LIN {X 0,Y 183.796,Z 363.678,A -85,B 0,C 180,E1 7701.816,E2 7701.816} C_VEL
LIN {X 0,Y 180.44,Z 378.523,A -85,B 0,C 180,E1 7700.122,E2 7700.122} C_VEL
LIN {X 0,Y 176.218,Z 391.784,A -85,B 0,C 180,E1 7698.008,E2 7698.008} C_VEL
LIN {X 0,Y 171.582,Z 403.279,A -85,B 0,C 180,E1 7695.544,E2 7695.544} C_VEL
LIN {X 0,Y 166.647,Z 413.424,A -85,B 0,C 180,E1 7692.682,E2 7692.682} C_VEL
LIN {X 0,Y 161.304,Z 422.653,A -85,B 0,C 180,E1 7689.21,E2 7689.21} C_VEL
LIN {X 0,Y 156.045,Z 430.534,A -85,B 0,C 180,E1 7685.213,E2 7685.213} C_VEL
LIN {X 0,Y 150.742,Z 437.424,A -85,B 0,C 180,E1 7680.268,E2 7680.268} C_VEL
LIN {X 0,Y 146.163,Z 442.505,A -85,B 0,C 180,E1 7674.659,E2 7674.659} C_VEL
LIN {X 0,Y 142.797,Z 445.543,A -85,B 0,C 180,E1 7668.786,E2 7668.786} C_VEL
LIN {X 0,Y 140.665,Z 446.734,A -85,B 0,C 180,E1 7662.726,E2 7662.726} C_VEL
LIN {X 0,Y 139.739,Z 446.152,A -85,B 0,C 180,E1 7656.571,E2 7656.571} C_VEL
LIN {X 0,Y 140.025,Z 443.543,A -85,B 0,C 180,E1 7649.997,E2 7649.997} C_VEL
LIN {X 0,Y 141.478,Z 439.126,A -85,B 0,C 180,E1 7643.912,E2 7643.912} C_VEL
LIN {X 0,Y 143.867,Z 433.071,A -85,B 0,C 180,E1 7638.37,E2 7638.37} C_VEL
LIN {X 0,Y 146.979,Z 425.519,A -85,B 0,C 180,E1 7633.396,E2 7633.396} C_VEL
LIN {X 0,Y 147.344,Z 424.201,A -85,B 0,C 180,E1 7632.625,E2 7632.625} C_VEL
LIN {X 0,Y 145.87,Z 423.422,A -85,B 0,C 180,E1 7631.533,E2 7631.533} C_VEL
LIN {X 0,Y 141.985,Z 433.557,A -85,B 0,C 180,E1 7624.342,E2 7624.342} C_VEL
LIN {X 0,Y 140.16,Z 439.981,A -85,B 0,C 180,E1 7618.095,E2 7618.095} C_VEL
LIN {X 0,Y 139.61,Z 444.799,A -85,B 0,C 180,E1 7611.456,E2 7611.456} C_VEL
LIN {X 0,Y 140.498,Z 447.794,A -85,B 0,C 180,E1 7604.627,E2 7604.627} C_VEL
LIN {X 0,Y 143.009,Z 449.031,A -85,B 0,C 180,E1 7597.807,E2 7597.807} C_VEL
LIN {X 0,Y 146.933,Z 448.501,A -85,B 0,C 180,E1 7591.6,E2 7591.6} C_VEL
LIN {X 0,Y 152.727,Z 446.052,A -85,B 0,C 180,E1 7585.381,E2 7585.381} C_VEL
LIN {X 0,Y 160,Z 441.734,A -85,B 0,C 180,E1 7579.723,E2 7579.723} C_VEL
LIN {X 0,Y 168.194,Z 435.599,A -85,B 0,C 180,E1 7574.811,E2 7574.811} C_VEL
LIN {X 0,Y 176.992,Z 427.833,A -85,B 0,C 180,E1 7570.586,E2 7570.586} C_VEL
LIN {X 0,Y 185.661,Z 418.872,A -85,B 0,C 180,E1 7567.116,E2 7567.116} C_VEL
LIN {X 0,Y 194.986,Z 407.509,A -85,B 0,C 180,E1 7563.936,E2 7563.936} C_VEL
LIN {X 0,Y 203.524,Z 395.312,A -85,B 0,C 180,E1 7561.408,E2 7561.408} C_VEL
LIN {X 0,Y 210.985,Z 382.54,A -85,B 0,C 180,E1 7559.417,E2 7559.417} C_VEL
LIN {X 0,Y 218.224,Z 367.365,A -85,B 0,C 180,E1 7557.637,E2 7557.637} C_VEL
LIN {X 0,Y 224.14,Z 351.874,A -85,B 0,C 180,E1 7556.279,E2 7556.279} C_VEL
LIN {X 0,Y 228.785,Z 335.328,A -85,B 0,C 180,E1 7555.225,E2 7555.225} C_VEL
LIN {X 0,Y 232.053,Z 318.038,A -85,B 0,C 180,E1 7554.464,E2 7554.464} C_VEL
LIN {X 0,Y 241.488,Z 250.304,A -85,B 0,C 180,E1 7552.506,E2 7552.506} C_VEL
LIN {X 0,Y 240.741,Z 246.563,A -85,B 0,C 180,E1 7550.498,E2 7550.498} C_VEL
LIN {X 0,Y 240.162,Z 243.632,A -85,B 0,C 180,E1 7548.351,E2 7548.351} C_VEL
LIN {X 0,Y 239.883,Z 241.404,A -85,B 0,C 180,E1 7545.243,E2 7545.243} C_VEL
LIN {X 0,Y 240.273,Z 241.241,A -85,B 0,C 180,E1 7542.065,E2 7542.065} C_VEL
LIN {X 0,Y 241.515,Z 243.115,A -85,B 0,C 180,E1 7538.635,E2 7538.635} C_VEL
LIN {X 0,Y 242.511,Z 245.708,A -85,B 0,C 180,E1 7536.743,E2 7536.743} C_VEL
LIN {X 0,Y 230.891,Z 333.654,A -85,B 0,C 180,E1 7534.471,E2 7534.471} C_VEL
LIN {X 0,Y 227.213,Z 350.101,A -85,B 0,C 180,E1 7533.868,E2 7533.868} C_VEL
LIN {X 0,Y 224.792,Z 357.503,A -85,B 0,C 180,E1 7533.772,E2 7533.772} C_VEL
LIN {X 0,Y 217.369,Z 373.68,A -85,B 0,C 180,E1 7534.209,E2 7534.209} C_VEL
LIN {X 0,Y 213.861,Z 380.585,A -85,B 0,C 180,E1 7534.095,E2 7534.095} C_VEL
LIN {X 0,Y 212.895,Z 382.52,A -85,B 0,C 180,E1 7533.967,E2 7533.967} C_VEL
LIN {X 0,Y 204.588,Z 398.255,A -85,B 0,C 180,E1 7532.504,E2 7532.504} C_VEL
LIN {X 0,Y 195.17,Z 413.15,A -85,B 0,C 180,E1 7530.568,E2 7530.568} C_VEL
LIN {X 0,Y 184.964,Z 426.922,A -85,B 0,C 180,E1 7528.073,E2 7528.073} C_VEL
LIN {X 0,Y 174.557,Z 439.14,A -85,B 0,C 180,E1 7524.998,E2 7524.998} C_VEL
LIN {X 0,Y 163.56,Z 450.596,A -85,B 0,C 180,E1 7520.932,E2 7520.932} C_VEL
LIN {X 0,Y 153.123,Z 460.494,A -85,B 0,C 180,E1 7515.915,E2 7515.915} C_VEL
LIN {X 0,Y 144.228,Z 468.323,A -85,B 0,C 180,E1 7510.148,E2 7510.148} C_VEL
LIN {X 0,Y 136.834,Z 474.713,A -85,B 0,C 180,E1 7503.235,E2 7503.235} C_VEL
LIN {X 0,Y 131.616,Z 479.56,A -85,B 0,C 180,E1 7495.18,E2 7495.18} C_VEL
LIN {X 0,Y 129.261,Z 482.628,A -85,B 0,C 180,E1 7486.433,E2 7486.433} C_VEL
LIN {X 0,Y 129.758,Z 483.716,A -85,B 0,C 180,E1 7477.976,E2 7477.976} C_VEL
LIN {X 0,Y 131.875,Z 483.304,A -85,B 0,C 180,E1 7470.438,E2 7470.438} C_VEL
LIN {X 0,Y 130.994,Z 483.773,A -85,B 0,C 180,E1 7466.941,E2 7466.941} C_VEL
LIN {X 0,Y 129.415,Z 483.078,A -85,B 0,C 180,E1 7460.217,E2 7460.217} C_VEL
LIN {X 0,Y 129.295,Z 480.56,A -85,B 0,C 180,E1 7453.378,E2 7453.378} C_VEL
LIN {X 0,Y 130.92,Z 476.166,A -85,B 0,C 180,E1 7446.605,E2 7446.605} C_VEL
LIN {X 0,Y 134.304,Z 469.671,A -85,B 0,C 180,E1 7440.084,E2 7440.084} C_VEL
LIN {X 0,Y 138.579,Z 462.091,A -85,B 0,C 180,E1 7434.75,E2 7434.75} C_VEL
LIN {X 0,Y 143.545,Z 453.197,A -85,B 0,C 180,E1 7430.152,E2 7430.152} C_VEL
LIN {X 0,Y 149.389,Z 441.861,A -85,B 0,C 180,E1 7425.893,E2 7425.893} C_VEL
LIN {X 0,Y 155.141,Z 429.09,A -85,B 0,C 180,E1 7422.45,E2 7422.45} C_VEL
LIN {X 0,Y 159.866,Z 416.561,A -85,B 0,C 180,E1 7419.995,E2 7419.995} C_VEL
LIN {X 0,Y 163.873,Z 403.35,A -85,B 0,C 180,E1 7418.092,E2 7418.092} C_VEL
LIN {X 0,Y 167.255,Z 387.828,A -85,B 0,C 180,E1 7416.541,E2 7416.541} C_VEL
LIN {X 0,Y 169.352,Z 371.857,A -85,B 0,C 180,E1 7415.588,E2 7415.588} C_VEL
LIN {X 0,Y 170.942,Z 353.783,A -85,B 0,C 180,E1 7414.832,E2 7414.832} C_VEL
LIN {X 0,Y 173.502,Z 335.522,A -85,B 0,C 180,E1 7413.757,E2 7413.757} C_VEL
LIN {X 0,Y 181.035,Z 244.738,A -85,B 0,C 180,E1 7410.511,E2 7410.511} C_VEL
LIN {X 0,Y 191.3,Z 201.884,A -85,B 0,C 180,E1 7407.552,E2 7407.552} C_VEL
LIN {X 0,Y 189.274,Z 188.28,A -85,B 0,C 180,E1 7402.682,E2 7402.682} C_VEL
LIN {X 0,Y 187.949,Z 177.866,A -85,B 0,C 180,E1 7398.132,E2 7398.132} C_VEL
LIN {X 0,Y 187.052,Z 175.913,A -85,B 0,C 180,E1 7396.138,E2 7396.138} C_VEL
LIN {X 0,Y 184.12,Z 171.648,A -85,B 0,C 180,E1 7387.174,E2 7387.174} C_VEL
LIN {X 0,Y 183.556,Z 171.776,A -85,B 0,C 180,E1 7383.747,E2 7383.747} C_VEL
LIN {X 0,Y 183.965,Z 175.013,A -85,B 0,C 180,E1 7375.323,E2 7375.323} C_VEL
LIN {X 0,Y 185.238,Z 179.369,A -85,B 0,C 180,E1 7370.367,E2 7370.367} C_VEL
LIN {X 0,Y 186.45,Z 183.613,A -85,B 0,C 180,E1 7366.667,E2 7366.667} C_VEL
LIN {X 0,Y 188.095,Z 189.403,A -85,B 0,C 180,E1 7362.681,E2 7362.681} C_VEL
LIN {X 0,Y 189.901,Z 196.74,A -85,B 0,C 180,E1 7358.697,E2 7358.697} C_VEL
LIN {X 0,Y 191.572,Z 205.206,A -85,B 0,C 180,E1 7354.99,E2 7354.99} C_VEL
LIN {X 0,Y 192.499,Z 212.026,A -85,B 0,C 180,E1 7352.541,E2 7352.541} C_VEL
LIN {X 0,Y 188.599,Z 232.595,A -85,B 0,C 180,E1 7349.437,E2 7349.437} C_VEL
LIN {X 0,Y 188.915,Z 240.844,A -85,B 0,C 180,E1 7348.727,E2 7348.727} C_VEL
LIN {X 0,Y 182.567,Z 320.837,A -85,B 0,C 180,E1 7346.205,E2 7346.205} C_VEL
LIN {X 0,Y 180.809,Z 349.598,A -85,B 0,C 180,E1 7344.905,E2 7344.905} C_VEL
LIN {X 0,Y 178.761,Z 364.13,A -85,B 0,C 180,E1 7343.782,E2 7343.782} C_VEL
LIN {X 0,Y 175.424,Z 378.468,A -85,B 0,C 180,E1 7342.163,E2 7342.163} C_VEL
LIN {X 0,Y 171.236,Z 391.377,A -85,B 0,C 180,E1 7340.155,E2 7340.155} C_VEL
LIN {X 0,Y 166.342,Z 403.249,A -85,B 0,C 180,E1 7337.67,E2 7337.67} C_VEL
LIN {X 0,Y 160.841,Z 414.076,A -85,B 0,C 180,E1 7334.62,E2 7334.62} C_VEL
LIN {X 0,Y 155.136,Z 423.474,A -85,B 0,C 180,E1 7331.054,E2 7331.054} C_VEL
LIN {X 0,Y 149.57,Z 431.381,A -85,B 0,C 180,E1 7326.983,E2 7326.983} C_VEL
LIN {X 0,Y 143.88,Z 438.33,A -85,B 0,C 180,E1 7321.876,E2 7321.876} C_VEL
LIN {X 0,Y 139.217,Z 443.189,A -85,B 0,C 180,E1 7316.438,E2 7316.438} C_VEL
LIN {X 0,Y 135.535,Z 446.37,A -85,B 0,C 180,E1 7310.46,E2 7310.46} C_VEL
LIN {X 0,Y 133.01,Z 447.81,A -85,B 0,C 180,E1 7303.915,E2 7303.915} C_VEL
LIN {X 0,Y 131.832,Z 447.296,A -85,B 0,C 180,E1 7296.967,E2 7296.967} C_VEL
LIN {X 0,Y 132.082,Z 444.737,A -85,B 0,C 180,E1 7289.997,E2 7289.997} C_VEL
LIN {X 0,Y 133.597,Z 440.371,A -85,B 0,C 180,E1 7283.551,E2 7283.551} C_VEL
LIN {X 0,Y 136.123,Z 434.384,A -85,B 0,C 180,E1 7277.698,E2 7277.698} C_VEL
LIN {X 0,Y 139.286,Z 427.144,A -85,B 0,C 180,E1 7272.609,E2 7272.609} C_VEL
LIN {X 0,Y 137.358,Z 426.181,A -85,B 0,C 180,E1 7271.141,E2 7271.141} C_VEL
LIN {X 0,Y 133.913,Z 434.986,A -85,B 0,C 180,E1 7264.335,E2 7264.335} C_VEL
LIN {X 0,Y 132.028,Z 441.741,A -85,B 0,C 180,E1 7257.207,E2 7257.207} C_VEL
LIN {X 0,Y 131.693,Z 446.225,A -85,B 0,C 180,E1 7250.372,E2 7250.372} C_VEL
LIN {X 0,Y 132.906,Z 449.118,A -85,B 0,C 180,E1 7243.132,E2 7243.132} C_VEL
LIN {X 0,Y 135.887,Z 450.266,A -85,B 0,C 180,E1 7235.96,E2 7235.96} C_VEL
LIN {X 0,Y 140.709,Z 449.5,A -85,B 0,C 180,E1 7229.066,E2 7229.066} C_VEL
LIN {X 0,Y 147.342,Z 446.84,A -85,B 0,C 180,E1 7222.642,E2 7222.642} C_VEL
LIN {X 0,Y 154.93,Z 442.571,A -85,B 0,C 180,E1 7217.221,E2 7217.221} C_VEL
LIN {X 0,Y 163.752,Z 436.36,A -85,B 0,C 180,E1 7212.318,E2 7212.318} C_VEL
LIN {X 0,Y 173.27,Z 428.382,A -85,B 0,C 180,E1 7208.078,E2 7208.078} C_VEL
LIN {X 0,Y 182.575,Z 419.158,A -85,B 0,C 180,E1 7204.633,E2 7204.633} C_VEL
LIN {X 0,Y 192.056,Z 408.086,A -85,B 0,C 180,E1 7201.643,E2 7201.643} C_VEL
LIN {X 0,Y 201.142,Z 395.526,A -85,B 0,C 180,E1 7199.146,E2 7199.146} C_VEL
LIN {X 0,Y 209.233,Z 382.045,A -85,B 0,C 180,E1 7197.151,E2 7197.151} C_VEL
LIN {X 0,Y 216.649,Z 366.908,A -85,B 0,C 180,E1 7195.475,E2 7195.475} C_VEL
LIN {X 0,Y 222.539,Z 351.55,A -85,B 0,C 180,E1 7194.211,E2 7194.211} C_VEL
LIN {X 0,Y 227.291,Z 334.726,A -85,B 0,C 180,E1 7193.203,E2 7193.203} C_VEL
LIN {X 0,Y 230.555,Z 317.53,A -85,B 0,C 180,E1 7192.492,E2 7192.492} C_VEL
LIN {X 0,Y 239.48,Z 255.386,A -85,B 0,C 180,E1 7190.75,E2 7190.75} C_VEL
LIN {X 0,Y 238.842,Z 251.44,A -85,B 0,C 180,E1 7188.041,E2 7188.041} C_VEL
LIN {X 0,Y 238.655,Z 249.244,A -85,B 0,C 180,E1 7184.945,E2 7184.945} C_VEL
LIN {X 0,Y 239.067,Z 249.206,A -85,B 0,C 180,E1 7181.972,E2 7181.972} C_VEL
LIN {X 0,Y 240.17,Z 250.984,A -85,B 0,C 180,E1 7178.881,E2 7178.881} C_VEL
LIN {X 0,Y 240.303,Z 251.671,A -85,B 0,C 180,E1 7178.473,E2 7178.473} C_VEL
LIN {X 0,Y 229.224,Z 332.504,A -85,B 0,C 180,E1 7176.449,E2 7176.449} C_VEL
LIN {X 0,Y 224.869,Z 350.985,A -85,B 0,C 180,E1 7175.796,E2 7175.796} C_VEL
LIN {X 0,Y 219.099,Z 368.129,A -85,B 0,C 180,E1 7174.941,E2 7174.941} C_VEL
LIN {X 0,Y 212.895,Z 382.52,A -85,B 0,C 180,E1 7173.967,E2 7173.967} C_VEL
LIN {X 0,Y 209.155,Z 389.39,A -85,B 0,C 180,E1 7173.651,E2 7173.651} C_VEL
LIN {X 0,Y 198.862,Z 403.987,A -85,B 0,C 180,E1 7173.579,E2 7173.579} C_VEL
LIN {X 0,Y 194.314,Z 410.036,A -85,B 0,C 180,E1 7173.203,E2 7173.203} C_VEL
LIN {X 0,Y 193.113,Z 411.695,A -85,B 0,C 180,E1 7172.995,E2 7172.995} C_VEL
LIN {X 0,Y 183.25,Z 424.637,A -85,B 0,C 180,E1 7170.812,E2 7170.812} C_VEL
LIN {X 0,Y 172.328,Z 437.018,A -85,B 0,C 180,E1 7167.901,E2 7167.901} C_VEL
LIN {X 0,Y 160.652,Z 448.602,A -85,B 0,C 180,E1 7164.01,E2 7164.01} C_VEL
LIN {X 0,Y 150.025,Z 458.061,A -85,B 0,C 180,E1 7159.447,E2 7159.447} C_VEL
LIN {X 0,Y 139.614,Z 466.571,A -85,B 0,C 180,E1 7153.437,E2 7153.437} C_VEL
LIN {X 0,Y 131.208,Z 473.061,A -85,B 0,C 180,E1 7146.473,E2 7146.473} C_VEL
LIN {X 0,Y 124.945,Z 478,A -85,B 0,C 180,E1 7138.177,E2 7138.177} C_VEL
LIN {X 0,Y 121.653,Z 481.153,A -85,B 0,C 180,E1 7129.062,E2 7129.062} C_VEL
LIN {X 0,Y 121.494,Z 482.433,A -85,B 0,C 180,E1 7119.955,E2 7119.955} C_VEL
LIN {X 0,Y 123.521,Z 481.958,A -85,B 0,C 180,E1 7111.859,E2 7111.859} C_VEL
LIN {X 0,Y 123.844,Z 482.358,A -85,B 0,C 180,E1 7109.541,E2 7109.541} C_VEL
LIN {X 0,Y 121.921,Z 482.518,A -85,B 0,C 180,E1 7102.938,E2 7102.938} C_VEL
LIN {X 0,Y 121.188,Z 480.901,A -85,B 0,C 180,E1 7095.673,E2 7095.673} C_VEL
LIN {X 0,Y 122.25,Z 477.411,A -85,B 0,C 180,E1 7088.409,E2 7088.409} C_VEL
LIN {X 0,Y 124.954,Z 472.42,A -85,B 0,C 180,E1 7081.833,E2 7081.833} C_VEL
LIN {X 0,Y 129.243,Z 465.518,A -85,B 0,C 180,E1 7075.62,E2 7075.62} C_VEL
LIN {X 0,Y 134.533,Z 457.053,A -85,B 0,C 180,E1 7070.276,E2 7070.276} C_VEL
LIN {X 0,Y 139.88,Z 448.042,A -85,B 0,C 180,E1 7066.109,E2 7066.109} C_VEL
LIN {X 0,Y 145.909,Z 436.717,A -85,B 0,C 180,E1 7062.267,E2 7062.267} C_VEL
LIN {X 0,Y 151.602,Z 424.223,A -85,B 0,C 180,E1 7059.206,E2 7059.206} C_VEL
LIN {X 0,Y 156.414,Z 411.487,A -85,B 0,C 180,E1 7056.932,E2 7056.932} C_VEL
LIN {X 0,Y 160.678,Z 396.975,A -85,B 0,C 180,E1 7055.092,E2 7055.092} C_VEL
LIN {X 0,Y 163.805,Z 381.683,A -85,B 0,C 180,E1 7053.824,E2 7053.824} C_VEL
LIN {X 0,Y 165.534,Z 365.855,A -85,B 0,C 180,E1 7053.019,E2 7053.019} C_VEL
LIN {X 0,Y 174.621,Z 255.346,A -85,B 0,C 180,E1 7049.006,E2 7049.006} C_VEL
LIN {X 0,Y 187.079,Z 205.346,A -85,B 0,C 180,E1 7045.558,E2 7045.558} C_VEL
LIN {X 0,Y 185.622,Z 193.516,A -85,B 0,C 180,E1 7041.155,E2 7041.155} C_VEL
LIN {X 0,Y 184.931,Z 184.749,A -85,B 0,C 180,E1 7037.218,E2 7037.218} C_VEL
LIN {X 0,Y 184.057,Z 183.174,A -85,B 0,C 180,E1 7035.437,E2 7035.437} C_VEL
LIN {X 0,Y 181.483,Z 179.183,A -85,B 0,C 180,E1 7026.961,E2 7026.961} C_VEL
LIN {X 0,Y 180.96,Z 179.369,A -85,B 0,C 180,E1 7023.801,E2 7023.801} C_VEL
LIN {X 0,Y 181.161,Z 182.294,A -85,B 0,C 180,E1 7015.885,E2 7015.885} C_VEL
LIN {X 0,Y 181.959,Z 186.551,A -85,B 0,C 180,E1 7010.83,E2 7010.83} C_VEL
LIN {X 0,Y 183.046,Z 190.826,A -85,B 0,C 180,E1 7007.058,E2 7007.058} C_VEL
LIN {X 0,Y 184.708,Z 197.276,A -85,B 0,C 180,E1 7002.678,E2 7002.678} C_VEL
LIN {X 0,Y 186.345,Z 205.722,A -85,B 0,C 180,E1 6998.27,E2 6998.27} C_VEL
LIN {X 0,Y 187.814,Z 215.098,A -85,B 0,C 180,E1 6994.454,E2 6994.454} C_VEL
LIN {X 0,Y 187.708,Z 216.611,A -85,B 0,C 180,E1 6994.1,E2 6994.1} C_VEL
LIN {X 0,Y 184.249,Z 233.796,A -85,B 0,C 180,E1 6991.496,E2 6991.496} C_VEL
LIN {X 0,Y 184.478,Z 242.195,A -85,B 0,C 180,E1 6990.756,E2 6990.756} C_VEL
LIN {X 0,Y 177.922,Z 321.341,A -85,B 0,C 180,E1 6988.269,E2 6988.269} C_VEL
LIN {X 0,Y 175.985,Z 350.749,A -85,B 0,C 180,E1 6986.926,E2 6986.926} C_VEL
LIN {X 0,Y 173.789,Z 365.423,A -85,B 0,C 180,E1 6985.78,E2 6985.78} C_VEL
LIN {X 0,Y 170.243,Z 379.828,A -85,B 0,C 180,E1 6984.138,E2 6984.138} C_VEL
LIN {X 0,Y 165.892,Z 392.552,A -85,B 0,C 180,E1 6982.139,E2 6982.139} C_VEL
LIN {X 0,Y 160.777,Z 404.347,A -85,B 0,C 180,E1 6979.647,E2 6979.647} C_VEL
LIN {X 0,Y 154.671,Z 415.715,A -85,B 0,C 180,E1 6976.382,E2 6976.382} C_VEL
LIN {X 0,Y 148.189,Z 425.663,A -85,B 0,C 180,E1 6972.427,E2 6972.427} C_VEL
LIN {X 0,Y 142.025,Z 433.686,A -85,B 0,C 180,E1 6967.954,E2 6967.954} C_VEL
LIN {X 0,Y 136.352,Z 440.055,A -85,B 0,C 180,E1 6962.859,E2 6962.859} C_VEL
LIN {X 0,Y 131.47,Z 444.731,A -85,B 0,C 180,E1 6957.145,E2 6957.145} C_VEL
LIN {X 0,Y 127.541,Z 447.754,A -85,B 0,C 180,E1 6950.653,E2 6950.653} C_VEL
LIN {X 0,Y 125.019,Z 448.929,A -85,B 0,C 180,E1 6943.879,E2 6943.879} C_VEL
LIN {X 0,Y 123.898,Z 448.331,A -85,B 0,C 180,E1 6936.949,E2 6936.949} C_VEL
LIN {X 0,Y 124.137,Z 445.923,A -85,B 0,C 180,E1 6929.996,E2 6929.996} C_VEL
LIN {X 0,Y 125.722,Z 441.617,A -85,B 0,C 180,E1 6923.145,E2 6923.145} C_VEL
LIN {X 0,Y 128.172,Z 436.197,A -85,B 0,C 180,E1 6917.38,E2 6917.38} C_VEL
LIN {X 0,Y 131.024,Z 429.999,A -85,B 0,C 180,E1 6912.537,E2 6912.537} C_VEL
LIN {X 0,Y 128.849,Z 428.917,A -85,B 0,C 180,E1 6910.699,E2 6910.699} C_VEL
LIN {X 0,Y 125.198,Z 438.327,A -85,B 0,C 180,E1 6902.403,E2 6902.403} C_VEL
LIN {X 0,Y 123.794,Z 444.268,A -85,B 0,C 180,E1 6895.005,E2 6895.005} C_VEL
LIN {X 0,Y 124.027,Z 448.452,A -85,B 0,C 180,E1 6887.373,E2 6887.373} C_VEL
LIN {X 0,Y 126.048,Z 450.835,A -85,B 0,C 180,E1 6879.692,E2 6879.692} C_VEL
LIN {X 0,Y 130.142,Z 451.423,A -85,B 0,C 180,E1 6872.014,E2 6872.014} C_VEL
LIN {X 0,Y 135.91,Z 450.205,A -85,B 0,C 180,E1 6865.187,E2 6865.187} C_VEL
LIN {X 0,Y 143.046,Z 447.274,A -85,B 0,C 180,E1 6859.18,E2 6859.18} C_VEL
LIN {X 0,Y 152.158,Z 442.224,A -85,B 0,C 180,E1 6853.451,E2 6853.451} C_VEL
LIN {X 0,Y 161.852,Z 435.547,A -85,B 0,C 180,E1 6848.718,E2 6848.718} C_VEL
LIN {X 0,Y 172.127,Z 426.993,A -85,B 0,C 180,E1 6844.665,E2 6844.665} C_VEL
LIN {X 0,Y 182.034,Z 417.242,A -85,B 0,C 180,E1 6841.414,E2 6841.414} C_VEL
LIN {X 0,Y 191.295,Z 406.5,A -85,B 0,C 180,E1 6838.803,E2 6838.803} C_VEL
LIN {X 0,Y 200.339,Z 394.02,A -85,B 0,C 180,E1 6836.551,E2 6836.551} C_VEL
LIN {X 0,Y 208.268,Z 380.879,A -85,B 0,C 180,E1 6834.767,E2 6834.767} C_VEL
LIN {X 0,Y 215.454,Z 366.393,A -85,B 0,C 180,E1 6833.28,E2 6833.28} C_VEL
LIN {X 0,Y 221.477,Z 350.826,A -85,B 0,C 180,E1 6832.086,E2 6832.086} C_VEL
LIN {X 0,Y 226.316,Z 333.886,A -85,B 0,C 180,E1 6831.14,E2 6831.14} C_VEL
LIN {X 0,Y 229.524,Z 316.629,A -85,B 0,C 180,E1 6830.48,E2 6830.48} C_VEL
LIN {X 0,Y 237.686,Z 260.927,A -85,B 0,C 180,E1 6828.966,E2 6828.966} C_VEL
LIN {X 0,Y 237.472,Z 258.67,A -85,B 0,C 180,E1 6827.106,E2 6827.106} C_VEL
LIN {X 0,Y 237.454,Z 257.086,A -85,B 0,C 180,E1 6824.617,E2 6824.617} C_VEL
LIN {X 0,Y 237.866,Z 257.176,A -85,B 0,C 180,E1 6821.878,E2 6821.878} C_VEL
LIN {X 0,Y 238.377,Z 258.15,A -85,B 0,C 180,E1 6820.226,E2 6820.226} C_VEL
LIN {X 0,Y 227.756,Z 331.961,A -85,B 0,C 180,E1 6818.438,E2 6818.438} C_VEL
LIN {X 0,Y 223.304,Z 350.351,A -85,B 0,C 180,E1 6817.825,E2 6817.825} C_VEL
LIN {X 0,Y 217.682,Z 366.751,A -85,B 0,C 180,E1 6817.066,E2 6817.066} C_VEL
LIN {X 0,Y 210.219,Z 383.339,A -85,B 0,C 180,E1 6815.997,E2 6815.997} C_VEL
LIN {X 0,Y 201.492,Z 399.008,A -85,B 0,C 180,E1 6814.576,E2 6814.576} C_VEL
LIN {X 0,Y 193.113,Z 411.695,A -85,B 0,C 180,E1 6812.995,E2 6812.995} C_VEL
LIN {X 0,Y 188.453,Z 417.576,A -85,B 0,C 180,E1 6812.379,E2 6812.379} C_VEL
LIN {X 0,Y 175.895,Z 430.053,A -85,B 0,C 180,E1 6811.576,E2 6811.576} C_VEL
LIN {X 0,Y 170.489,Z 435.097,A -85,B 0,C 180,E1 6810.801,E2 6810.801} C_VEL
LIN {X 0,Y 169.071,Z 436.456,A -85,B 0,C 180,E1 6810.462,E2 6810.462} C_VEL
LIN {X 0,Y 157.353,Z 447.46,A -85,B 0,C 180,E1 6806.876,E2 6806.876} C_VEL
LIN {X 0,Y 145.527,Z 457.295,A -85,B 0,C 180,E1 6802.2,E2 6802.2} C_VEL
LIN {X 0,Y 134.926,Z 465.259,A -85,B 0,C 180,E1 6796.574,E2 6796.574} C_VEL
LIN {X 0,Y 125.28,Z 471.932,A -85,B 0,C 180,E1 6789.273,E2 6789.273} C_VEL
LIN {X 0,Y 118.048,Z 476.88,A -85,B 0,C 180,E1 6780.547,E2 6780.547} C_VEL
LIN {X 0,Y 114.074,Z 479.921,A -85,B 0,C 180,E1 6771.065,E2 6771.065} C_VEL
LIN {X 0,Y 113.437,Z 481.14,A -85,B 0,C 180,E1 6761.185,E2 6761.185} C_VEL
LIN {X 0,Y 115.646,Z 480.715,A -85,B 0,C 180,E1 6751.49,E2 6751.49} C_VEL
LIN {X 0,Y 115.832,Z 481.201,A -85,B 0,C 180,E1 6749.509,E2 6749.509} C_VEL
LIN {X 0,Y 113.845,Z 481.403,A -85,B 0,C 180,E1 6742.434,E2 6742.434} C_VEL
LIN {X 0,Y 113.28,Z 479.655,A -85,B 0,C 180,E1 6734.125,E2 6734.125} C_VEL
LIN {X 0,Y 114.97,Z 475.799,A -85,B 0,C 180,E1 6725.879,E2 6725.879} C_VEL
LIN {X 0,Y 118.645,Z 470.137,A -85,B 0,C 180,E1 6718.505,E2 6718.505} C_VEL
LIN {X 0,Y 123.344,Z 463.429,A -85,B 0,C 180,E1 6712.563,E2 6712.563} C_VEL
LIN {X 0,Y 129.301,Z 454.745,A -85,B 0,C 180,E1 6707.124,E2 6707.124} C_VEL
LIN {X 0,Y 135.771,Z 444.461,A -85,B 0,C 180,E1 6702.578,E2 6702.578} C_VEL
LIN {X 0,Y 141.778,Z 433.677,A -85,B 0,C 180,E1 6699.133,E2 6699.133} C_VEL
LIN {X 0,Y 147.598,Z 421.499,A -85,B 0,C 180,E1 6696.287,E2 6696.287} C_VEL
LIN {X 0,Y 153.059,Z 407.35,A -85,B 0,C 180,E1 6693.946,E2 6693.946} C_VEL
LIN {X 0,Y 157.103,Z 393.489,A -85,B 0,C 180,E1 6692.349,E2 6692.349} C_VEL
LIN {X 0,Y 160.023,Z 378.996,A -85,B 0,C 180,E1 6691.211,E2 6691.211} C_VEL
LIN {X 0,Y 162.035,Z 360.125,A -85,B 0,C 180,E1 6690.369,E2 6690.369} C_VEL
LIN {X 0,Y 171.075,Z 254.844,A -85,B 0,C 180,E1 6686.6,E2 6686.6} C_VEL
LIN {X 0,Y 183.097,Z 208.863,A -85,B 0,C 180,E1 6683.493,E2 6683.493} C_VEL
LIN {X 0,Y 182.077,Z 197.953,A -85,B 0,C 180,E1 6679.237,E2 6679.237} C_VEL
LIN {X 0,Y 181.813,Z 191.577,A -85,B 0,C 180,E1 6676.288,E2 6676.288} C_VEL
LIN {X 0,Y 180.924,Z 190.272,A -85,B 0,C 180,E1 6674.399,E2 6674.399} C_VEL
LIN {X 0,Y 178.707,Z 186.672,A -85,B 0,C 180,E1 6666.747,E2 6666.747} C_VEL
LIN {X 0,Y 178.163,Z 186.896,A -85,B 0,C 180,E1 6663.861,E2 6663.861} C_VEL
LIN {X 0,Y 178.024,Z 189.756,A -85,B 0,C 180,E1 6656.098,E2 6656.098} C_VEL
LIN {X 0,Y 178.674,Z 193.721,A -85,B 0,C 180,E1 6651.309,E2 6651.309} C_VEL
LIN {X 0,Y 179.768,Z 198.403,A -85,B 0,C 180,E1 6647.145,E2 6647.145} C_VEL
LIN {X 0,Y 181.257,Z 205.324,A -85,B 0,C 180,E1 6642.669,E2 6642.669} C_VEL
LIN {X 0,Y 182.538,Z 213.323,A -85,B 0,C 180,E1 6638.61,E2 6638.61} C_VEL
LIN {X 0,Y 183.353,Z 219.875,A -85,B 0,C 180,E1 6635.943,E2 6635.943} C_VEL
LIN {X 0,Y 180.141,Z 234.838,A -85,B 0,C 180,E1 6633.668,E2 6633.668} C_VEL
LIN {X 0,Y 180.295,Z 243.443,A -85,B 0,C 180,E1 6632.885,E2 6632.885} C_VEL
LIN {X 0,Y 173.525,Z 321.807,A -85,B 0,C 180,E1 6630.443,E2 6630.443} C_VEL
LIN {X 0,Y 171.417,Z 351.696,A -85,B 0,C 180,E1 6629.071,E2 6629.071} C_VEL
LIN {X 0,Y 169.008,Z 366.865,A -85,B 0,C 180,E1 6627.879,E2 6627.879} C_VEL
LIN {X 0,Y 165.292,Z 381.139,A -85,B 0,C 180,E1 6626.241,E2 6626.241} C_VEL
LIN {X 0,Y 160.597,Z 394.122,A -85,B 0,C 180,E1 6624.18,E2 6624.18} C_VEL
LIN {X 0,Y 155.039,Z 406.155,A -85,B 0,C 180,E1 6621.582,E2 6621.582} C_VEL
LIN {X 0,Y 148.658,Z 417.336,A -85,B 0,C 180,E1 6618.289,E2 6618.289} C_VEL
LIN {X 0,Y 141.83,Z 427.174,A -85,B 0,C 180,E1 6614.255,E2 6614.255} C_VEL
LIN {X 0,Y 135.128,Z 435.297,A -85,B 0,C 180,E1 6609.515,E2 6609.515} C_VEL
LIN {X 0,Y 129.279,Z 441.369,A -85,B 0,C 180,E1 6604.369,E2 6604.369} C_VEL
LIN {X 0,Y 124.068,Z 445.983,A -85,B 0,C 180,E1 6598.386,E2 6598.386} C_VEL
LIN {X 0,Y 119.631,Z 449.078,A -85,B 0,C 180,E1 6591.058,E2 6591.058} C_VEL
LIN {X 0,Y 116.908,Z 450.062,A -85,B 0,C 180,E1 6583.347,E2 6583.347} C_VEL
LIN {X 0,Y 115.915,Z 449.127,A -85,B 0,C 180,E1 6575.937,E2 6575.937} C_VEL
LIN {X 0,Y 116.33,Z 446.661,A -85,B 0,C 180,E1 6569.011,E2 6569.011} C_VEL
LIN {X 0,Y 118.188,Z 442.168,A -85,B 0,C 180,E1 6561.728,E2 6561.728} C_VEL
LIN {X 0,Y 121.208,Z 436.009,A -85,B 0,C 180,E1 6555.18,E2 6555.18} C_VEL
LIN {X 0,Y 122.706,Z 432.762,A -85,B 0,C 180,E1 6552.437,E2 6552.437} C_VEL
LIN {X 0,Y 120.337,Z 431.482,A -85,B 0,C 180,E1 6550.206,E2 6550.206} C_VEL
LIN {X 0,Y 117.03,Z 439.927,A -85,B 0,C 180,E1 6541.968,E2 6541.968} C_VEL
LIN {X 0,Y 115.764,Z 445.749,A -85,B 0,C 180,E1 6534.029,E2 6534.029} C_VEL
LIN {X 0,Y 116.296,Z 449.841,A -85,B 0,C 180,E1 6525.857,E2 6525.857} C_VEL
LIN {X 0,Y 118.794,Z 452.11,A -85,B 0,C 180,E1 6517.7,E2 6517.7} C_VEL
LIN {X 0,Y 123.597,Z 452.627,A -85,B 0,C 180,E1 6509.57,E2 6509.57} C_VEL
LIN {X 0,Y 129.986,Z 451.324,A -85,B 0,C 180,E1 6502.618,E2 6502.618} C_VEL
LIN {X 0,Y 138.421,Z 448.067,A -85,B 0,C 180,E1 6496.109,E2 6496.109} C_VEL
LIN {X 0,Y 147.602,Z 443.317,A -85,B 0,C 180,E1 6490.806,E2 6490.806} C_VEL
LIN {X 0,Y 157.777,Z 436.71,A -85,B 0,C 180,E1 6486.185,E2 6486.185} C_VEL
LIN {X 0,Y 169.161,Z 427.73,A -85,B 0,C 180,E1 6482.033,E2 6482.033} C_VEL
LIN {X 0,Y 179.511,Z 418.003,A -85,B 0,C 180,E1 6478.915,E2 6478.915} C_VEL
LIN {X 0,Y 189.889,Z 406.245,A -85,B 0,C 180,E1 6476.228,E2 6476.228} C_VEL
LIN {X 0,Y 199.606,Z 393.15,A -85,B 0,C 180,E1 6474.036,E2 6474.036} C_VEL
LIN {X 0,Y 207.819,Z 379.691,A -85,B 0,C 180,E1 6472.362,E2 6472.362} C_VEL
LIN {X 0,Y 215.14,Z 364.757,A -85,B 0,C 180,E1 6470.972,E2 6470.972} C_VEL
LIN {X 0,Y 221.303,Z 348.587,A -85,B 0,C 180,E1 6469.852,E2 6469.852} C_VEL
LIN {X 0,Y 225.859,Z 332.139,A -85,B 0,C 180,E1 6469.027,E2 6469.027} C_VEL
LIN {X 0,Y 229.319,Z 312.475,A -85,B 0,C 180,E1 6468.359,E2 6468.359} C_VEL
LIN {X 0,Y 236.219,Z 266.796,A -85,B 0,C 180,E1 6467.161,E2 6467.161} C_VEL
LIN {X 0,Y 236.24,Z 264.987,A -85,B 0,C 180,E1 6464.536,E2 6464.536} C_VEL
LIN {X 0,Y 236.62,Z 265.089,A -85,B 0,C 180,E1 6461.996,E2 6461.996} C_VEL
LIN {X 0,Y 226.782,Z 331.219,A -85,B 0,C 180,E1 6460.462,E2 6460.462} C_VEL
LIN {X 0,Y 222.147,Z 349.696,A -85,B 0,C 180,E1 6459.887,E2 6459.887} C_VEL
LIN {X 0,Y 216.12,Z 366.584,A -85,B 0,C 180,E1 6459.156,E2 6459.156} C_VEL
LIN {X 0,Y 208.437,Z 383.045,A -85,B 0,C 180,E1 6458.16,E2 6458.16} C_VEL
LIN {X 0,Y 199.552,Z 398.526,A -85,B 0,C 180,E1 6456.846,E2 6456.846} C_VEL
LIN {X 0,Y 189.582,Z 412.927,A -85,B 0,C 180,E1 6455.115,E2 6455.115} C_VEL
LIN {X 0,Y 178.668,Z 426.199,A -85,B 0,C 180,E1 6452.851,E2 6452.851} C_VEL
LIN {X 0,Y 169.071,Z 436.456,A -85,B 0,C 180,E1 6450.462,E2 6450.462} C_VEL
LIN {X 0,Y 163.693,Z 441.237,A -85,B 0,C 180,E1 6449.381,E2 6449.381} C_VEL
LIN {X 0,Y 150.517,Z 450.423,A -85,B 0,C 180,E1 6447.61,E2 6447.61} C_VEL
LIN {X 0,Y 144.669,Z 454.229,A -85,B 0,C 180,E1 6446.33,E2 6446.33} C_VEL
LIN {X 0,Y 142.478,Z 455.771,A -85,B 0,C 180,E1 6445.569,E2 6445.569} C_VEL
LIN {X 0,Y 130.681,Z 463.966,A -85,B 0,C 180,E1 6439.921,E2 6439.921} C_VEL
LIN {X 0,Y 120.384,Z 470.424,A -85,B 0,C 180,E1 6432.93,E2 6432.93} C_VEL
LIN {X 0,Y 112.075,Z 475.344,A -85,B 0,C 180,E1 6424.201,E2 6424.201} C_VEL
LIN {X 0,Y 106.947,Z 478.47,A -85,B 0,C 180,E1 6414.294,E2 6414.294} C_VEL
LIN {X 0,Y 105.383,Z 479.828,A -85,B 0,C 180,E1 6403.725,E2 6403.725} C_VEL
LIN {X 0,Y 107.17,Z 479.322,A -85,B 0,C 180,E1 6393.213,E2 6393.213} C_VEL
LIN {X 0,Y 107.983,Z 479.965,A -85,B 0,C 180,E1 6390.004,E2 6390.004} C_VEL
LIN {X 0,Y 105.871,Z 480.324,A -85,B 0,C 180,E1 6382.406,E2 6382.406} C_VEL
LIN {X 0,Y 105.32,Z 478.879,A -85,B 0,C 180,E1 6374.024,E2 6374.024} C_VEL
LIN {X 0,Y 106.917,Z 475.633,A -85,B 0,C 180,E1 6365.707,E2 6365.707} C_VEL
LIN {X 0,Y 110.694,Z 470.472,A -85,B 0,C 180,E1 6357.802,E2 6357.802} C_VEL
LIN {X 0,Y 116.461,Z 463.118,A -85,B 0,C 180,E1 6350.562,E2 6350.562} C_VEL
LIN {X 0,Y 123.404,Z 453.909,A -85,B 0,C 180,E1 6344.526,E2 6344.526} C_VEL
LIN {X 0,Y 130.372,Z 443.714,A -85,B 0,C 180,E1 6339.928,E2 6339.928} C_VEL
LIN {X 0,Y 137.116,Z 432.442,A -85,B 0,C 180,E1 6336.322,E2 6336.322} C_VEL
LIN {X 0,Y 143.307,Z 420.247,A -85,B 0,C 180,E1 6333.521,E2 6333.521} C_VEL
LIN {X 0,Y 149.077,Z 406.071,A -85,B 0,C 180,E1 6331.232,E2 6331.232} C_VEL
LIN {X 0,Y 153.319,Z 392.152,A -85,B 0,C 180,E1 6329.667,E2 6329.667} C_VEL
LIN {X 0,Y 156.426,Z 377.415,A -85,B 0,C 180,E1 6328.567,E2 6328.567} C_VEL
LIN {X 0,Y 158.555,Z 358.436,A -85,B 0,C 180,E1 6327.766,E2 6327.766} C_VEL
LIN {X 0,Y 168.048,Z 253.526,A -85,B 0,C 180,E1 6324.043,E2 6324.043} C_VEL
LIN {X 0,Y 179.343,Z 212.448,A -85,B 0,C 180,E1 6321.34,E2 6321.34} C_VEL
LIN {X 0,Y 178.726,Z 202.443,A -85,B 0,C 180,E1 6317.247,E2 6317.247} C_VEL
LIN {X 0,Y 178.68,Z 198.299,A -85,B 0,C 180,E1 6315.248,E2 6315.248} C_VEL
LIN {X 0,Y 175.892,Z 194.152,A -85,B 0,C 180,E1 6306.527,E2 6306.527} C_VEL
LIN {X 0,Y 175.259,Z 194.516,A -85,B 0,C 180,E1 6303.597,E2 6303.597} C_VEL
LIN {X 0,Y 175.042,Z 196.925,A -85,B 0,C 180,E1 6296.725,E2 6296.725} C_VEL
LIN {X 0,Y 175.629,Z 200.982,A -85,B 0,C 180,E1 6291.817,E2 6291.817} C_VEL
LIN {X 0,Y 176.52,Z 205.332,A -85,B 0,C 180,E1 6287.902,E2 6287.902} C_VEL
LIN {X 0,Y 177.617,Z 212.257,A -85,B 0,C 180,E1 6283.315,E2 6283.315} C_VEL
LIN {X 0,Y 178.624,Z 220.146,A -85,B 0,C 180,E1 6279.35,E2 6279.35} C_VEL
LIN {X 0,Y 179.021,Z 223.87,A -85,B 0,C 180,E1 6277.765,E2 6277.765} C_VEL
LIN {X 0,Y 176.307,Z 236.037,A -85,B 0,C 180,E1 6275.922,E2 6275.922} C_VEL
LIN {X 0,Y 176.377,Z 244.641,A -85,B 0,C 180,E1 6275.113,E2 6275.113} C_VEL
LIN {X 0,Y 169.392,Z 322.252,A -85,B 0,C 180,E1 6272.728,E2 6272.728} C_VEL
LIN {X 0,Y 167.076,Z 352.862,A -85,B 0,C 180,E1 6271.316,E2 6271.316} C_VEL
LIN {X 0,Y 164.733,Z 367.046,A -85,B 0,C 180,E1 6270.214,E2 6270.214} C_VEL
LIN {X 0,Y 160.988,Z 381.138,A -85,B 0,C 180,E1 6268.641,E2 6268.641} C_VEL
LIN {X 0,Y 156.542,Z 393.328,A -85,B 0,C 180,E1 6266.789,E2 6266.789} C_VEL
LIN {X 0,Y 150.513,Z 406.118,A -85,B 0,C 180,E1 6264.133,E2 6264.133} C_VEL
LIN {X 0,Y 143.759,Z 417.523,A -85,B 0,C 180,E1 6260.844,E2 6260.844} C_VEL
LIN {X 0,Y 136.784,Z 427.194,A -85,B 0,C 180,E1 6256.963,E2 6256.963} C_VEL
LIN {X 0,Y 130.097,Z 435.043,A -85,B 0,C 180,E1 6252.551,E2 6252.551} C_VEL
LIN {X 0,Y 123.206,Z 441.905,A -85,B 0,C 180,E1 6246.903,E2 6246.903} C_VEL
LIN {X 0,Y 117.088,Z 446.96,A -85,B 0,C 180,E1 6240.248,E2 6240.248} C_VEL
LIN {X 0,Y 112.455,Z 449.966,A -85,B 0,C 180,E1 6233.025,E2 6233.025} C_VEL
LIN {X 0,Y 109.587,Z 451.11,A -85,B 0,C 180,E1 6225.881,E2 6225.881} C_VEL
LIN {X 0,Y 108.105,Z 450.613,A -85,B 0,C 180,E1 6217.97,E2 6217.97} C_VEL
LIN {X 0,Y 108.315,Z 448.087,A -85,B 0,C 180,E1 6209.467,E2 6209.467} C_VEL
LIN {X 0,Y 110.166,Z 443.761,A -85,B 0,C 180,E1 6201.646,E2 6201.646} C_VEL
LIN {X 0,Y 113.032,Z 438.32,A -85,B 0,C 180,E1 6195.132,E2 6195.132} C_VEL
LIN {X 0,Y 114.495,Z 435.474,A -85,B 0,C 180,E1 6192.436,E2 6192.436} C_VEL
LIN {X 0,Y 111.792,Z 434.049,A -85,B 0,C 180,E1 6189.582,E2 6189.582} C_VEL
LIN {X 0,Y 108.534,Z 442.626,A -85,B 0,C 180,E1 6179.995,E2 6179.995} C_VEL
LIN {X 0,Y 107.765,Z 447.956,A -85,B 0,C 180,E1 6171.56,E2 6171.56} C_VEL
LIN {X 0,Y 108.972,Z 451.628,A -85,B 0,C 180,E1 6162.765,E2 6162.765} C_VEL
LIN {X 0,Y 112.406,Z 453.602,A -85,B 0,C 180,E1 6154.084,E2 6154.084} C_VEL
LIN {X 0,Y 117.981,Z 453.74,A -85,B 0,C 180,E1 6146.056,E2 6146.056} C_VEL
LIN {X 0,Y 125.948,Z 451.985,A -85,B 0,C 180,E1 6138.516,E2 6138.516} C_VEL
LIN {X 0,Y 135.107,Z 448.552,A -85,B 0,C 180,E1 6132.337,E2 6132.337} C_VEL
LIN {X 0,Y 145.303,Z 443.327,A -85,B 0,C 180,E1 6127.116,E2 6127.116} C_VEL
LIN {X 0,Y 156.688,Z 436.112,A -85,B 0,C 180,E1 6122.561,E2 6122.561} C_VEL
LIN {X 0,Y 168.012,Z 427.341,A -85,B 0,C 180,E1 6118.897,E2 6118.897} C_VEL
LIN {X 0,Y 179.456,Z 416.63,A -85,B 0,C 180,E1 6115.821,E2 6115.821} C_VEL
LIN {X 0,Y 189.764,Z 405.139,A -85,B 0,C 180,E1 6113.455,E2 6113.455} C_VEL
LIN {X 0,Y 199.14,Z 392.537,A -85,B 0,C 180,E1 6111.546,E2 6111.546} C_VEL
LIN {X 0,Y 208.22,Z 377.578,A -85,B 0,C 180,E1 6109.871,E2 6109.871} C_VEL
LIN {X 0,Y 215.736,Z 362.132,A -85,B 0,C 180,E1 6108.593,E2 6108.593} C_VEL
LIN {X 0,Y 221.676,Z 345.959,A -85,B 0,C 180,E1 6107.604,E2 6107.604} C_VEL
LIN {X 0,Y 226.18,Z 328.647,A -85,B 0,C 180,E1 6106.845,E2 6106.845} C_VEL
LIN {X 0,Y 231.197,Z 297.573,A -85,B 0,C 180,E1 6105.981,E2 6105.981} C_VEL
LIN {X 0,Y 234.907,Z 273.45,A -85,B 0,C 180,E1 6105.393,E2 6105.393} C_VEL
LIN {X 0,Y 235.106,Z 272.755,A -85,B 0,C 180,E1 6103.783,E2 6103.783} C_VEL
LIN {X 0,Y 226.115,Z 330.546,A -85,B 0,C 180,E1 6102.5,E2 6102.5} C_VEL
LIN {X 0,Y 221.228,Z 349.423,A -85,B 0,C 180,E1 6101.957,E2 6101.957} C_VEL
LIN {X 0,Y 214.904,Z 366.56,A -85,B 0,C 180,E1 6101.272,E2 6101.272} C_VEL
LIN {X 0,Y 207.026,Z 382.919,A -85,B 0,C 180,E1 6100.356,E2 6100.356} C_VEL
LIN {X 0,Y 197.937,Z 398.154,A -85,B 0,C 180,E1 6099.153,E2 6099.153} C_VEL
LIN {X 0,Y 187.701,Z 412.331,A -85,B 0,C 180,E1 6097.554,E2 6097.554} C_VEL
LIN {X 0,Y 176.872,Z 425.082,A -85,B 0,C 180,E1 6095.528,E2 6095.528} C_VEL
LIN {X 0,Y 164.754,Z 437.304,A -85,B 0,C 180,E1 6092.755,E2 6092.755} C_VEL
LIN {X 0,Y 152.475,Z 448.059,A -85,B 0,C 180,E1 6089.213,E2 6089.213} C_VEL
LIN {X 0,Y 142.478,Z 455.771,A -85,B 0,C 180,E1 6085.569,E2 6085.569} C_VEL
LIN {X 0,Y 137.024,Z 459.251,A -85,B 0,C 180,E1 6083.802,E2 6083.802} C_VEL
LIN {X 0,Y 122.742,Z 465.889,A -85,B 0,C 180,E1 6080.047,E2 6080.047} C_VEL
LIN {X 0,Y 116.94,Z 468.482,A -85,B 0,C 180,E1 6077.481,E2 6077.481} C_VEL
LIN {X 0,Y 115.996,Z 468.946,A -85,B 0,C 180,E1 6076.849,E2 6076.849} C_VEL
LIN {X 0,Y 106.614,Z 473.826,A -85,B 0,C 180,E1 6068.245,E2 6068.245} C_VEL
LIN {X 0,Y 100.203,Z 477.022,A -85,B 0,C 180,E1 6057.973,E2 6057.973} C_VEL
LIN {X 0,Y 97.536,Z 478.474,A -85,B 0,C 180,E1 6046.685,E2 6046.685} C_VEL
LIN {X 0,Y 98.66,Z 478.105,A -85,B 0,C 180,E1 6035.238,E2 6035.238} C_VEL
LIN {X 0,Y 99.269,Z 478.032,A -85,B 0,C 180,E1 6032.891,E2 6032.891} C_VEL
LIN {X 0,Y 99.95,Z 478.812,A -85,B 0,C 180,E1 6030.004,E2 6030.004} C_VEL
LIN {X 0,Y 97.704,Z 479.166,A -85,B 0,C 180,E1 6021.175,E2 6021.175} C_VEL
LIN {X 0,Y 97.572,Z 477.484,A -85,B 0,C 180,E1 6011.483,E2 6011.483} C_VEL
LIN {X 0,Y 99.921,Z 474.021,A -85,B 0,C 180,E1 6002.599,E2 6002.599} C_VEL
LIN {X 0,Y 104.176,Z 469.065,A -85,B 0,C 180,E1 5994.845,E2 5994.845} C_VEL
LIN {X 0,Y 110.222,Z 462.198,A -85,B 0,C 180,E1 5987.84,E2 5987.84} C_VEL
LIN {X 0,Y 117.205,Z 453.788,A -85,B 0,C 180,E1 5982.089,E2 5982.089} C_VEL
LIN {X 0,Y 124.623,Z 443.907,A -85,B 0,C 180,E1 5977.419,E2 5977.419} C_VEL
LIN {X 0,Y 132.103,Z 432.431,A -85,B 0,C 180,E1 5973.645,E2 5973.645} C_VEL
LIN {X 0,Y 139.201,Z 419.354,A -85,B 0,C 180,E1 5970.662,E2 5970.662} C_VEL
LIN {X 0,Y 145.051,Z 405.781,A -85,B 0,C 180,E1 5968.501,E2 5968.501} C_VEL
LIN {X 0,Y 149.51,Z 392.25,A -85,B 0,C 180,E1 5966.994,E2 5966.994} C_VEL
LIN {X 0,Y 152.989,Z 377.082,A -85,B 0,C 180,E1 5965.876,E2 5965.876} C_VEL
LIN {X 0,Y 155.233,Z 358.651,A -85,B 0,C 180,E1 5965.109,E2 5965.109} C_VEL
LIN {X 0,Y 165.374,Z 252.248,A -85,B 0,C 180,E1 5961.404,E2 5961.404} C_VEL
LIN {X 0,Y 175.75,Z 216.009,A -85,B 0,C 180,E1 5959.094,E2 5959.094} C_VEL
LIN {X 0,Y 175.649,Z 205.51,A -85,B 0,C 180,E1 5954.504,E2 5954.504} C_VEL
LIN {X 0,Y 173.239,Z 201.694,A -85,B 0,C 180,E1 5946.295,E2 5946.295} C_VEL
LIN {X 0,Y 172.474,Z 202.44,A -85,B 0,C 180,E1 5942.657,E2 5942.657} C_VEL
LIN {X 0,Y 172.353,Z 204.515,A -85,B 0,C 180,E1 5937.006,E2 5937.006} C_VEL
LIN {X 0,Y 172.607,Z 208.243,A -85,B 0,C 180,E1 5932.343,E2 5932.343} C_VEL
LIN {X 0,Y 173.159,Z 212.635,A -85,B 0,C 180,E1 5928.34,E2 5928.34} C_VEL
LIN {X 0,Y 173.915,Z 218.648,A -85,B 0,C 180,E1 5924.323,E2 5924.323} C_VEL
LIN {X 0,Y 174.652,Z 225.91,A -85,B 0,C 180,E1 5920.606,E2 5920.606} C_VEL
LIN {X 0,Y 174.805,Z 228.168,A -85,B 0,C 180,E1 5919.627,E2 5919.627} C_VEL
LIN {X 0,Y 172.756,Z 237.173,A -85,B 0,C 180,E1 5918.28,E2 5918.28} C_VEL
LIN {X 0,Y 172.734,Z 245.863,A -85,B 0,C 180,E1 5917.438,E2 5917.438} C_VEL
LIN {X 0,Y 165.547,Z 322.689,A -85,B 0,C 180,E1 5915.124,E2 5915.124} C_VEL
LIN {X 0,Y 163.023,Z 353.918,A -85,B 0,C 180,E1 5913.685,E2 5913.685} C_VEL
LIN {X 0,Y 160.427,Z 368.719,A -85,B 0,C 180,E1 5912.534,E2 5912.534} C_VEL
LIN {X 0,Y 156.347,Z 383.08,A -85,B 0,C 180,E1 5910.919,E2 5910.919} C_VEL
LIN {X 0,Y 151.217,Z 396.085,A -85,B 0,C 180,E1 5908.893,E2 5908.893} C_VEL
LIN {X 0,Y 145.262,Z 407.885,A -85,B 0,C 180,E1 5906.387,E2 5906.387} C_VEL
LIN {X 0,Y 138.176,Z 419.162,A -85,B 0,C 180,E1 5903.086,E2 5903.086} C_VEL
LIN {X 0,Y 130.826,Z 428.706,A -85,B 0,C 180,E1 5899.161,E2 5899.161} C_VEL
LIN {X 0,Y 123.748,Z 436.449,A -85,B 0,C 180,E1 5894.658,E2 5894.658} C_VEL
LIN {X 0,Y 116.899,Z 442.818,A -85,B 0,C 180,E1 5889.261,E2 5889.261} C_VEL
LIN {X 0,Y 110.247,Z 447.931,A -85,B 0,C 180,E1 5882.345,E2 5882.345} C_VEL
LIN {X 0,Y 105.14,Z 450.999,A -85,B 0,C 180,E1 5874.731,E2 5874.731} C_VEL
LIN {X 0,Y 101.76,Z 452.215,A -85,B 0,C 180,E1 5866.551,E2 5866.551} C_VEL
LIN {X 0,Y 100.172,Z 451.654,A -85,B 0,C 180,E1 5858.028,E2 5858.028} C_VEL
LIN {X 0,Y 100.448,Z 449.061,A -85,B 0,C 180,E1 5848.855,E2 5848.855} C_VEL
LIN {X 0,Y 102.521,Z 444.66,A -85,B 0,C 180,E1 5840.452,E2 5840.452} C_VEL
LIN {X 0,Y 105.978,Z 438.63,A -85,B 0,C 180,E1 5832.99,E2 5832.99} C_VEL
LIN {X 0,Y 106.195,Z 438.043,A -85,B 0,C 180,E1 5832.333,E2 5832.333} C_VEL
LIN {X 0,Y 103.263,Z 436.465,A -85,B 0,C 180,E1 5828.889,E2 5828.889} C_VEL
LIN {X 0,Y 100.338,Z 444.384,A -85,B 0,C 180,E1 5818.982,E2 5818.982} C_VEL
LIN {X 0,Y 99.896,Z 449.695,A -85,B 0,C 180,E1 5809.41,E2 5809.41} C_VEL
LIN {X 0,Y 101.845,Z 453.278,A -85,B 0,C 180,E1 5799.654,E2 5799.654} C_VEL
LIN {X 0,Y 106.169,Z 454.934,A -85,B 0,C 180,E1 5790.569,E2 5790.569} C_VEL
LIN {X 0,Y 113.32,Z 454.771,A -85,B 0,C 180,E1 5781.753,E2 5781.753} C_VEL
LIN {X 0,Y 121.947,Z 452.834,A -85,B 0,C 180,E1 5774.638,E2 5774.638} C_VEL
LIN {X 0,Y 132.747,Z 448.784,A -85,B 0,C 180,E1 5768.229,E2 5768.229} C_VEL
LIN {X 0,Y 144.2,Z 443.08,A -85,B 0,C 180,E1 5763.13,E2 5763.13} C_VEL
LIN {X 0,Y 156.007,Z 435.629,A -85,B 0,C 180,E1 5758.992,E2 5758.992} C_VEL
LIN {X 0,Y 168.077,Z 426.374,A -85,B 0,C 180,E1 5755.565,E2 5755.565} C_VEL
LIN {X 0,Y 179.357,Z 415.959,A -85,B 0,C 180,E1 5752.894,E2 5752.894} C_VEL
LIN {X 0,Y 190.53,Z 403.433,A -85,B 0,C 180,E1 5750.611,E2 5750.611} C_VEL
LIN {X 0,Y 200.648,Z 389.702,A -85,B 0,C 180,E1 5748.794,E2 5748.794} C_VEL
LIN {X 0,Y 208.984,Z 375.778,A -85,B 0,C 180,E1 5747.431,E2 5747.431} C_VEL
LIN {X 0,Y 216.399,Z 360.029,A -85,B 0,C 180,E1 5746.28,E2 5746.28} C_VEL
LIN {X 0,Y 222.367,Z 343.411,A -85,B 0,C 180,E1 5745.383,E2 5745.383} C_VEL
LIN {X 0,Y 226.53,Z 326.721,A -85,B 0,C 180,E1 5744.738,E2 5744.738} C_VEL
LIN {X 0,Y 226.89,Z 324.706,A -85,B 0,C 180,E1 5744.663,E2 5744.663} C_VEL
LIN {X 0,Y 222.761,Z 342.624,A -85,B 0,C 180,E1 5744.233,E2 5744.233} C_VEL
LIN {X 0,Y 217.193,Z 359.04,A -85,B 0,C 180,E1 5743.711,E2 5743.711} C_VEL
LIN {X 0,Y 209.669,Z 375.835,A -85,B 0,C 180,E1 5742.97,E2 5742.97} C_VEL
LIN {X 0,Y 200.812,Z 391.545,A -85,B 0,C 180,E1 5741.994,E2 5741.994} C_VEL
LIN {X 0,Y 190.709,Z 406.141,A -85,B 0,C 180,E1 5740.689,E2 5740.689} C_VEL
LIN {X 0,Y 179.017,Z 420.224,A -85,B 0,C 180,E1 5738.87,E2 5738.87} C_VEL
LIN {X 0,Y 166.783,Z 432.7,A -85,B 0,C 180,E1 5736.529,E2 5736.529} C_VEL
LIN {X 0,Y 154.167,Z 443.672,A -85,B 0,C 180,E1 5733.513,E2 5733.513} C_VEL
LIN {X 0,Y 141.439,Z 453.233,A -85,B 0,C 180,E1 5729.596,E2 5729.596} C_VEL
LIN {X 0,Y 128.768,Z 461.585,A -85,B 0,C 180,E1 5724.384,E2 5724.384} C_VEL
LIN {X 0,Y 117.375,Z 468.219,A -85,B 0,C 180,E1 5717.83,E2 5717.83} C_VEL
LIN {X 0,Y 115.996,Z 468.946,A -85,B 0,C 180,E1 5716.849,E2 5716.849} C_VEL
LIN {X 0,Y 111.172,Z 471.045,A -85,B 0,C 180,E1 5713.944,E2 5713.944} C_VEL
LIN {X 0,Y 99.799,Z 474.123,A -85,B 0,C 180,E1 5707.874,E2 5707.874} C_VEL
LIN {X 0,Y 94.868,Z 475.284,A -85,B 0,C 180,E1 5703.58,E2 5703.58} C_VEL
LIN {X 0,Y 93.86,Z 475.607,A -85,B 0,C 180,E1 5702.028,E2 5702.028} C_VEL
LIN {X 0,Y 89.878,Z 477.153,A -85,B 0,C 180,E1 5689.501,E2 5689.501} C_VEL
LIN {X 0,Y 90.353,Z 476.783,A -85,B 0,C 180,E1 5676.997,E2 5676.997} C_VEL
LIN {X 0,Y 91.058,Z 476.66,A -85,B 0,C 180,E1 5673.782,E2 5673.782} C_VEL
LIN {X 0,Y 91.896,Z 477.656,A -85,B 0,C 180,E1 5670.005,E2 5670.005} C_VEL
LIN {X 0,Y 89.642,Z 478.036,A -85,B 0,C 180,E1 5660.374,E2 5660.374} C_VEL
LIN {X 0,Y 89.817,Z 476.397,A -85,B 0,C 180,E1 5649.818,E2 5649.818} C_VEL
LIN {X 0,Y 92.681,Z 472.988,A -85,B 0,C 180,E1 5640.253,E2 5640.253} C_VEL
LIN {X 0,Y 97.546,Z 468.094,A -85,B 0,C 180,E1 5632.054,E2 5632.054} C_VEL
LIN {X 0,Y 104.806,Z 460.722,A -85,B 0,C 180,E1 5624.322,E2 5624.322} C_VEL
LIN {X 0,Y 113.146,Z 451.498,A -85,B 0,C 180,E1 5618.149,E2 5618.149} C_VEL
LIN {X 0,Y 121.242,Z 441.282,A -85,B 0,C 180,E1 5613.607,E2 5613.607} C_VEL
LIN {X 0,Y 128.527,Z 430.591,A -85,B 0,C 180,E1 5610.295,E2 5610.295} C_VEL
LIN {X 0,Y 135.814,Z 417.746,A -85,B 0,C 180,E1 5607.496,E2 5607.496} C_VEL
LIN {X 0,Y 142.137,Z 403.623,A -85,B 0,C 180,E1 5605.376,E2 5605.376} C_VEL
LIN {X 0,Y 147.062,Z 388.783,A -85,B 0,C 180,E1 5603.882,E2 5603.882} C_VEL
LIN {X 0,Y 150.367,Z 374.077,A -85,B 0,C 180,E1 5602.944,E2 5602.944} C_VEL
LIN {X 0,Y 152.774,Z 353.269,A -85,B 0,C 180,E1 5602.117,E2 5602.117} C_VEL
LIN {X 0,Y 163.066,Z 250.97,A -85,B 0,C 180,E1 5598.689,E2 5598.689} C_VEL
LIN {X 0,Y 172.403,Z 219.631,A -85,B 0,C 180,E1 5596.778,E2 5596.778} C_VEL
LIN {X 0,Y 172.567,Z 212.627,A -85,B 0,C 180,E1 5593.571,E2 5593.571} C_VEL
LIN {X 0,Y 170.579,Z 209.236,A -85,B 0,C 180,E1 5586.056,E2 5586.056} C_VEL
LIN {X 0,Y 169.425,Z 211.58,A -85,B 0,C 180,E1 5577.801,E2 5577.801} C_VEL
LIN {X 0,Y 169.409,Z 215.425,A -85,B 0,C 180,E1 5572.88,E2 5572.88} C_VEL
LIN {X 0,Y 169.92,Z 219.997,A -85,B 0,C 180,E1 5568.802,E2 5568.802} C_VEL
LIN {X 0,Y 170.531,Z 225.73,A -85,B 0,C 180,E1 5565.049,E2 5565.049} C_VEL
LIN {X 0,Y 170.824,Z 232.387,A -85,B 0,C 180,E1 5561.596,E2 5561.596} C_VEL
LIN {X 0,Y 169.51,Z 238.513,A -85,B 0,C 180,E1 5560.711,E2 5560.711} C_VEL
LIN {X 0,Y 169.388,Z 247.118,A -85,B 0,C 180,E1 5559.859,E2 5559.859} C_VEL
LIN {X 0,Y 161.994,Z 323.256,A -85,B 0,C 180,E1 5557.624,E2 5557.624} C_VEL
LIN {X 0,Y 159.265,Z 354.96,A -85,B 0,C 180,E1 5556.171,E2 5556.171} C_VEL
LIN {X 0,Y 156.581,Z 369.576,A -85,B 0,C 180,E1 5555.051,E2 5555.051} C_VEL
LIN {X 0,Y 152.458,Z 383.596,A -85,B 0,C 180,E1 5553.514,E2 5553.514} C_VEL
LIN {X 0,Y 147.262,Z 396.404,A -85,B 0,C 180,E1 5551.586,E2 5551.586} C_VEL
LIN {X 0,Y 140.977,Z 408.452,A -85,B 0,C 180,E1 5549.104,E2 5549.104} C_VEL
LIN {X 0,Y 133.164,Z 420.318,A -85,B 0,C 180,E1 5545.676,E2 5545.676} C_VEL
LIN {X 0,Y 125.08,Z 430.221,A -85,B 0,C 180,E1 5541.565,E2 5541.565} C_VEL
LIN {X 0,Y 117.584,Z 437.857,A -85,B 0,C 180,E1 5536.988,E2 5536.988} C_VEL
LIN {X 0,Y 110.287,Z 444.149,A -85,B 0,C 180,E1 5531.432,E2 5531.432} C_VEL
LIN {X 0,Y 103.145,Z 449.189,A -85,B 0,C 180,E1 5524.205,E2 5524.205} C_VEL
LIN {X 0,Y 97.621,Z 452.18,A -85,B 0,C 180,E1 5516.125,E2 5516.125} C_VEL
LIN {X 0,Y 94.134,Z 453.306,A -85,B 0,C 180,E1 5507.935,E2 5507.935} C_VEL
LIN {X 0,Y 92.293,Z 452.793,A -85,B 0,C 180,E1 5498.719,E2 5498.719} C_VEL
LIN {X 0,Y 92.505,Z 450.249,A -85,B 0,C 180,E1 5488.757,E2 5488.757} C_VEL
LIN {X 0,Y 94.711,Z 445.903,A -85,B 0,C 180,E1 5479.657,E2 5479.657} C_VEL
LIN {X 0,Y 98.023,Z 440.571,A -85,B 0,C 180,E1 5472.33,E2 5472.33} C_VEL
LIN {X 0,Y 94.716,Z 438.876,A -85,B 0,C 180,E1 5468.019,E2 5468.019} C_VEL
LIN {X 0,Y 92.076,Z 446.424,A -85,B 0,C 180,E1 5457.11,E2 5457.11} C_VEL
LIN {X 0,Y 92.211,Z 451.558,A -85,B 0,C 180,E1 5446.595,E2 5446.595} C_VEL
LIN {X 0,Y 94.795,Z 454.698,A -85,B 0,C 180,E1 5436.709,E2 5436.709} C_VEL
LIN {X 0,Y 100.384,Z 456.239,A -85,B 0,C 180,E1 5426.631,E2 5426.631} C_VEL
LIN {X 0,Y 108.307,Z 455.92,A -85,B 0,C 180,E1 5418.026,E2 5418.026} C_VEL
LIN {X 0,Y 118.228,Z 453.71,A -85,B 0,C 180,E1 5410.724,E2 5410.724} C_VEL
LIN {X 0,Y 129.435,Z 449.736,A -85,B 0,C 180,E1 5404.769,E2 5404.769} C_VEL
LIN {X 0,Y 141.986,Z 443.764,A -85,B 0,C 180,E1 5399.75,E2 5399.75} C_VEL
LIN {X 0,Y 154.385,Z 436.23,A -85,B 0,C 180,E1 5395.863,E2 5395.863} C_VEL
LIN {X 0,Y 166.568,Z 427.181,A -85,B 0,C 180,E1 5392.759,E2 5392.759} C_VEL
LIN {X 0,Y 178.099,Z 416.936,A -85,B 0,C 180,E1 5390.305,E2 5390.305} C_VEL
LIN {X 0,Y 188.896,Z 405.309,A -85,B 0,C 180,E1 5388.311,E2 5388.311} C_VEL
LIN {X 0,Y 199.413,Z 391.535,A -85,B 0,C 180,E1 5386.591,E2 5386.591} C_VEL
LIN {X 0,Y 208.394,Z 377.177,A -85,B 0,C 180,E1 5385.269,E2 5385.269} C_VEL
LIN {X 0,Y 208.948,Z 376.164,A -85,B 0,C 180,E1 5385.157,E2 5385.157} C_VEL
LIN {X 0,Y 199.942,Z 391.526,A -85,B 0,C 180,E1 5384.294,E2 5384.294} C_VEL
LIN {X 0,Y 189.64,Z 405.866,A -85,B 0,C 180,E1 5383.13,E2 5383.13} C_VEL
LIN {X 0,Y 177.676,Z 419.79,A -85,B 0,C 180,E1 5381.486,E2 5381.486} C_VEL
LIN {X 0,Y 165.535,Z 431.713,A -85,B 0,C 180,E1 5379.432,E2 5379.432} C_VEL
LIN {X 0,Y 152.452,Z 442.574,A -85,B 0,C 180,E1 5376.668,E2 5376.668} C_VEL
LIN {X 0,Y 138.317,Z 452.648,A -85,B 0,C 180,E1 5372.77,E2 5372.77} C_VEL
LIN {X 0,Y 125.157,Z 460.686,A -85,B 0,C 180,E1 5367.872,E2 5367.872} C_VEL
LIN {X 0,Y 112.676,Z 467.292,A -85,B 0,C 180,E1 5361.347,E2 5361.347} C_VEL
LIN {X 0,Y 101.75,Z 472.32,A -85,B 0,C 180,E1 5352.695,E2 5352.695} C_VEL
LIN {X 0,Y 93.86,Z 475.607,A -85,B 0,C 180,E1 5342.028,E2 5342.028} C_VEL
LIN {X 0,Y 90.88,Z 476.292,A -85,B 0,C 180,E1 5337.597,E2 5337.597} C_VEL
LIN {X 0,Y 83.84,Z 476.24,A -85,B 0,C 180,E1 5327.981,E2 5327.981} C_VEL
LIN {X 0,Y 81.951,Z 475.726,A -85,B 0,C 180,E1 5321.961,E2 5321.961} C_VEL
LIN {X 0,Y 81.993,Z 475.551,A -85,B 0,C 180,E1 5320.019,E2 5320.019} C_VEL
LIN {X 0,Y 82.849,Z 475.268,A -85,B 0,C 180,E1 5314.851,E2 5314.851} C_VEL
LIN {X 0,Y 83.824,Z 476.497,A -85,B 0,C 180,E1 5310.005,E2 5310.005} C_VEL
LIN {X 0,Y 81.593,Z 476.899,A -85,B 0,C 180,E1 5299.414,E2 5299.414} C_VEL
LIN {X 0,Y 82.016,Z 475.462,A -85,B 0,C 180,E1 5288.554,E2 5288.554} C_VEL
LIN {X 0,Y 85.302,Z 472.244,A -85,B 0,C 180,E1 5278.172,E2 5278.172} C_VEL
LIN {X 0,Y 91.184,Z 467.117,A -85,B 0,C 180,E1 5268.866,E2 5268.866} C_VEL
LIN {X 0,Y 99.269,Z 459.777,A -85,B 0,C 180,E1 5260.895,E2 5260.895} C_VEL
LIN {X 0,Y 107.586,Z 451.382,A -85,B 0,C 180,E1 5255.14,E2 5255.14} C_VEL
LIN {X 0,Y 115.424,Z 442.419,A -85,B 0,C 180,E1 5250.962,E2 5250.962} C_VEL
LIN {X 0,Y 123.831,Z 431.148,A -85,B 0,C 180,E1 5247.364,E2 5247.364} C_VEL
LIN {X 0,Y 131.45,Z 418.733,A -85,B 0,C 180,E1 5244.648,E2 5244.648} C_VEL
LIN {X 0,Y 137.66,Z 406.209,A -85,B 0,C 180,E1 5242.727,E2 5242.727} C_VEL
LIN {X 0,Y 143.154,Z 391.723,A -85,B 0,C 180,E1 5241.194,E2 5241.194} C_VEL
LIN {X 0,Y 147.264,Z 375.93,A -85,B 0,C 180,E1 5240.134,E2 5240.134} C_VEL
LIN {X 0,Y 149.655,Z 359.096,A -85,B 0,C 180,E1 5239.472,E2 5239.472} C_VEL
LIN {X 0,Y 161.022,Z 250.055,A -85,B 0,C 180,E1 5235.925,E2 5235.925} C_VEL
LIN {X 0,Y 169.294,Z 223.383,A -85,B 0,C 180,E1 5234.362,E2 5234.362} C_VEL
LIN {X 0,Y 169.458,Z 219.739,A -85,B 0,C 180,E1 5232.609,E2 5232.609} C_VEL
LIN {X 0,Y 167.758,Z 216.724,A -85,B 0,C 180,E1 5226.158,E2 5226.158} C_VEL
LIN {X 0,Y 166.56,Z 218.95,A -85,B 0,C 180,E1 5218.279,E2 5218.279} C_VEL
LIN {X 0,Y 166.55,Z 222.731,A -85,B 0,C 180,E1 5213.45,E2 5213.45} C_VEL
LIN {X 0,Y 166.901,Z 227.51,A -85,B 0,C 180,E1 5209.239,E2 5209.239} C_VEL
LIN {X 0,Y 167.045,Z 234.009,A -85,B 0,C 180,E1 5205.085,E2 5205.085} C_VEL
LIN {X 0,Y 166.987,Z 237.059,A -85,B 0,C 180,E1 5203.6,E2 5203.6} C_VEL
LIN {X 0,Y 166.567,Z 242.38,A -85,B 0,C 180,E1 5202.95,E2 5202.95} C_VEL
LIN {X 0,Y 166.366,Z 248.441,A -85,B 0,C 180,E1 5202.373,E2 5202.373} C_VEL
LIN {X 0,Y 158.775,Z 323.722,A -85,B 0,C 180,E1 5200.235,E2 5200.235} C_VEL
LIN {X 0,Y 155.823,Z 355.991,A -85,B 0,C 180,E1 5198.773,E2 5198.773} C_VEL
LIN {X 0,Y 152.995,Z 370.676,A -85,B 0,C 180,E1 5197.668,E2 5197.668} C_VEL
LIN {X 0,Y 148.658,Z 384.779,A -85,B 0,C 180,E1 5196.157,E2 5196.157} C_VEL
LIN {X 0,Y 143.183,Z 397.667,A -85,B 0,C 180,E1 5194.256,E2 5194.256} C_VEL
LIN {X 0,Y 136.626,Z 409.654,A -85,B 0,C 180,E1 5191.831,E2 5191.831} C_VEL
LIN {X 0,Y 128.812,Z 420.986,A -85,B 0,C 180,E1 5188.623,E2 5188.623} C_VEL
LIN {X 0,Y 120.954,Z 430.246,A -85,B 0,C 180,E1 5184.915,E2 5184.915} C_VEL
LIN {X 0,Y 112.915,Z 438.159,A -85,B 0,C 180,E1 5180.381,E2 5180.381} C_VEL
LIN {X 0,Y 104.417,Z 445.067,A -85,B 0,C 180,E1 5174.342,E2 5174.342} C_VEL
LIN {X 0,Y 96.628,Z 450.163,A -85,B 0,C 180,E1 5166.875,E2 5166.875} C_VEL
LIN {X 0,Y 90.511,Z 453.213,A -85,B 0,C 180,E1 5158.354,E2 5158.354} C_VEL
LIN {X 0,Y 86.36,Z 454.411,A -85,B 0,C 180,E1 5148.91,E2 5148.91} C_VEL
LIN {X 0,Y 84.362,Z 453.831,A -85,B 0,C 180,E1 5138.858,E2 5138.858} C_VEL
LIN {X 0,Y 84.653,Z 451.22,A -85,B 0,C 180,E1 5127.964,E2 5127.964} C_VEL
LIN {X 0,Y 87.155,Z 446.8,A -85,B 0,C 180,E1 5118.078,E2 5118.078} C_VEL
LIN {X 0,Y 89.625,Z 442.94,A -85,B 0,C 180,E1 5112.129,E2 5112.129} C_VEL
LIN {X 0,Y 86.156,Z 441.177,A -85,B 0,C 180,E1 5106.936,E2 5106.936} C_VEL
LIN {X 0,Y 83.925,Z 448.338,A -85,B 0,C 180,E1 5095.114,E2 5095.114} C_VEL
LIN {X 0,Y 84.641,Z 453.124,A -85,B 0,C 180,E1 5083.89,E2 5083.89} C_VEL
LIN {X 0,Y 88.184,Z 456.153,A -85,B 0,C 180,E1 5072.954,E2 5072.954} C_VEL
LIN {X 0,Y 94.502,Z 457.499,A -85,B 0,C 180,E1 5062.993,E2 5062.993} C_VEL
LIN {X 0,Y 103.239,Z 457.132,A -85,B 0,C 180,E1 5054.409,E2 5054.409} C_VEL
LIN {X 0,Y 114.289,Z 454.831,A -85,B 0,C 180,E1 5047.036,E2 5047.036} C_VEL
LIN {X 0,Y 126.113,Z 450.919,A -85,B 0,C 180,E1 5041.364,E2 5041.364} C_VEL
LIN {X 0,Y 138.98,Z 445.173,A -85,B 0,C 180,E1 5036.701,E2 5036.701} C_VEL
LIN {X 0,Y 152.6,Z 437.287,A -85,B 0,C 180,E1 5032.849,E2 5032.849} C_VEL
LIN {X 0,Y 165.541,Z 428.074,A -85,B 0,C 180,E1 5029.912,E2 5029.912} C_VEL
LIN {X 0,Y 177.503,Z 417.69,A -85,B 0,C 180,E1 5027.641,E2 5027.641} C_VEL
LIN {X 0,Y 189.561,Z 404.946,A -85,B 0,C 180,E1 5025.674,E2 5025.674} C_VEL
LIN {X 0,Y 177.647,Z 418.491,A -85,B 0,C 180,E1 5024.254,E2 5024.254} C_VEL
LIN {X 0,Y 164.722,Z 430.751,A -85,B 0,C 180,E1 5022.367,E2 5022.367} C_VEL
LIN {X 0,Y 151.218,Z 441.583,A -85,B 0,C 180,E1 5019.875,E2 5019.875} C_VEL
LIN {X 0,Y 137.332,Z 451.022,A -85,B 0,C 180,E1 5016.548,E2 5016.548} C_VEL
LIN {X 0,Y 122.584,Z 459.549,A -85,B 0,C 180,E1 5011.758,E2 5011.758} C_VEL
LIN {X 0,Y 109.139,Z 466.06,A -85,B 0,C 180,E1 5005.545,E2 5005.545} C_VEL
LIN {X 0,Y 96.996,Z 471.049,A -85,B 0,C 180,E1 4997.05,E2 4997.05} C_VEL
LIN {X 0,Y 87.454,Z 474.399,A -85,B 0,C 180,E1 4985.673,E2 4985.673} C_VEL
LIN {X 0,Y 82.473,Z 475.817,A -85,B 0,C 180,E1 4972.832,E2 4972.832} C_VEL
LIN {X 0,Y 81.993,Z 475.551,A -85,B 0,C 180,E1 4960.019,E2 4960.019} C_VEL
LIN {X 0,Y 81.555,Z 475.377,A -85,B 0,C 180,E1 4956.973,E2 4956.973} C_VEL
LIN {X 0,Y 79.069,Z 475.395,A -85,B 0,C 180,E1 4952.536,E2 4952.536} C_VEL
LIN {X 0,Y 74.417,Z 475.769,A -85,B 0,C 180,E1 4944.482,E2 4944.482} C_VEL
LIN {X 0,Y 74.143,Z 475.795,A -85,B 0,C 180,E1 4943.294,E2 4943.294} C_VEL
LIN {X 0,Y 73.615,Z 475.249,A -85,B 0,C 180,E1 4931.803,E2 4931.803} C_VEL
LIN {X 0,Y 76.464,Z 472.71,A -85,B 0,C 180,E1 4919.345,E2 4919.345} C_VEL
LIN {X 0,Y 82.637,Z 468.055,A -85,B 0,C 180,E1 4908.29,E2 4908.29} C_VEL
LIN {X 0,Y 90.877,Z 461.562,A -85,B 0,C 180,E1 4899.64,E2 4899.64} C_VEL
LIN {X 0,Y 99.481,Z 453.997,A -85,B 0,C 180,E1 4893.475,E2 4893.475} C_VEL
LIN {X 0,Y 108.677,Z 444.734,A -85,B 0,C 180,E1 4888.581,E2 4888.581} C_VEL
LIN {X 0,Y 117.838,Z 433.825,A -85,B 0,C 180,E1 4884.795,E2 4884.795} C_VEL
LIN {X 0,Y 126.159,Z 421.759,A -85,B 0,C 180,E1 4881.999,E2 4881.999} C_VEL
LIN {X 0,Y 133.02,Z 409.489,A -85,B 0,C 180,E1 4880.032,E2 4880.032} C_VEL
LIN {X 0,Y 139.138,Z 395.433,A -85,B 0,C 180,E1 4878.469,E2 4878.469} C_VEL
LIN {X 0,Y 143.947,Z 379.865,A -85,B 0,C 180,E1 4877.335,E2 4877.335} C_VEL
LIN {X 0,Y 146.901,Z 363.933,A -85,B 0,C 180,E1 4876.637,E2 4876.637} C_VEL
LIN {X 0,Y 159.358,Z 249.14,A -85,B 0,C 180,E1 4873.088,E2 4873.088} C_VEL
LIN {X 0,Y 166.417,Z 227.205,A -85,B 0,C 180,E1 4871.874,E2 4871.874} C_VEL
LIN {X 0,Y 165.09,Z 224.267,A -85,B 0,C 180,E1 4865.909,E2 4865.909} C_VEL
LIN {X 0,Y 163.884,Z 226.527,A -85,B 0,C 180,E1 4858.601,E2 4858.601} C_VEL
LIN {X 0,Y 163.687,Z 230.029,A -85,B 0,C 180,E1 4854.039,E2 4854.039} C_VEL
LIN {X 0,Y 163.667,Z 234.357,A -85,B 0,C 180,E1 4850.15,E2 4850.15} C_VEL
LIN {X 0,Y 163.713,Z 240.214,A -85,B 0,C 180,E1 4846.4,E2 4846.4} C_VEL
LIN {X 0,Y 164.021,Z 241.893,A -85,B 0,C 180,E1 4845.765,E2 4845.765} C_VEL
LIN {X 0,Y 163.704,Z 249.606,A -85,B 0,C 180,E1 4844.979,E2 4844.979} C_VEL
LIN {X 0,Y 155.9,Z 324.231,A -85,B 0,C 180,E1 4842.948,E2 4842.948} C_VEL
LIN {X 0,Y 152.718,Z 357.058,A -85,B 0,C 180,E1 4841.485,E2 4841.485} C_VEL
LIN {X 0,Y 149.662,Z 372.121,A -85,B 0,C 180,E1 4840.376,E2 4840.376} C_VEL
LIN {X 0,Y 145.18,Z 386.007,A -85,B 0,C 180,E1 4838.927,E2 4838.927} C_VEL
LIN {X 0,Y 139.474,Z 398.86,A -85,B 0,C 180,E1 4837.09,E2 4837.09} C_VEL
LIN {X 0,Y 132.651,Z 410.79,A -85,B 0,C 180,E1 4834.747,E2 4834.747} C_VEL
LIN {X 0,Y 124.44,Z 422.143,A -85,B 0,C 180,E1 4831.611,E2 4831.611} C_VEL
LIN {X 0,Y 115.798,Z 431.761,A -85,B 0,C 180,E1 4827.79,E2 4827.79} C_VEL
LIN {X 0,Y 107.297,Z 439.568,A -85,B 0,C 180,E1 4823.256,E2 4823.256} C_VEL
LIN {X 0,Y 98.237,Z 446.395,A -85,B 0,C 180,E1 4817.116,E2 4817.116} C_VEL
LIN {X 0,Y 89.843,Z 451.421,A -85,B 0,C 180,E1 4809.365,E2 4809.365} C_VEL
LIN {X 0,Y 83.178,Z 454.394,A -85,B 0,C 180,E1 4800.316,E2 4800.316} C_VEL
LIN {X 0,Y 78.617,Z 455.516,A -85,B 0,C 180,E1 4790.077,E2 4790.077} C_VEL
LIN {X 0,Y 76.431,Z 454.861,A -85,B 0,C 180,E1 4779.026,E2 4779.026} C_VEL
LIN {X 0,Y 76.714,Z 452.409,A -85,B 0,C 180,E1 4767.753,E2 4767.753} C_VEL
LIN {X 0,Y 79.413,Z 448.042,A -85,B 0,C 180,E1 4756.896,E2 4756.896} C_VEL
LIN {X 0,Y 81.316,Z 445.338,A -85,B 0,C 180,E1 4752.092,E2 4752.092} C_VEL
LIN {X 0,Y 77.625,Z 443.445,A -85,B 0,C 180,E1 4745.652,E2 4745.652} C_VEL
LIN {X 0,Y 75.871,Z 450.373,A -85,B 0,C 180,E1 4732.254,E2 4732.254} C_VEL
LIN {X 0,Y 77.612,Z 455.024,A -85,B 0,C 180,E1 4719.372,E2 4719.372} C_VEL
LIN {X 0,Y 82.748,Z 457.858,A -85,B 0,C 180,E1 4707.335,E2 4707.335} C_VEL
LIN {X 0,Y 90.935,Z 458.794,A -85,B 0,C 180,E1 4696.931,E2 4696.931} C_VEL
LIN {X 0,Y 102.015,Z 457.843,A -85,B 0,C 180,E1 4688.122,E2 4688.122} C_VEL
LIN {X 0,Y 114.248,Z 455.105,A -85,B 0,C 180,E1 4681.506,E2 4681.506} C_VEL
LIN {X 0,Y 127.242,Z 450.594,A -85,B 0,C 180,E1 4676.378,E2 4676.378} C_VEL
LIN {X 0,Y 141.297,Z 444.124,A -85,B 0,C 180,E1 4672.188,E2 4672.188} C_VEL
LIN {X 0,Y 154.82,Z 436.177,A -85,B 0,C 180,E1 4669.015,E2 4669.015} C_VEL
LIN {X 0,Y 168.733,Z 425.975,A -85,B 0,C 180,E1 4666.37,E2 4666.37} C_VEL
LIN {X 0,Y 170.291,Z 424.719,A -85,B 0,C 180,E1 4666.108,E2 4666.108} C_VEL
LIN {X 0,Y 155.984,Z 436.602,A -85,B 0,C 180,E1 4664.057,E2 4664.057} C_VEL
LIN {X 0,Y 141.414,Z 446.73,A -85,B 0,C 180,E1 4661.347,E2 4661.347} C_VEL
LIN {X 0,Y 126.514,Z 455.407,A -85,B 0,C 180,E1 4657.625,E2 4657.625} C_VEL
LIN {X 0,Y 111.663,Z 462.554,A -85,B 0,C 180,E1 4652.44,E2 4652.44} C_VEL
LIN {X 0,Y 97.523,Z 468.192,A -85,B 0,C 180,E1 4645.112,E2 4645.112} C_VEL
LIN {X 0,Y 85.776,Z 472.024,A -85,B 0,C 180,E1 4635.327,E2 4635.327} C_VEL
LIN {X 0,Y 77.534,Z 474.094,A -85,B 0,C 180,E1 4622.8,E2 4622.8} C_VEL
LIN {X 0,Y 73.944,Z 474.448,A -85,B 0,C 180,E1 4608.125,E2 4608.125} C_VEL
LIN {X 0,Y 74.612,Z 473.748,A -85,B 0,C 180,E1 4596.546,E2 4596.546} C_VEL
LIN {X 0,Y 75.734,Z 475.336,A -85,B 0,C 180,E1 4590.006,E2 4590.006} C_VEL
LIN {X 0,Y 74.143,Z 475.795,A -85,B 0,C 180,E1 4583.294,E2 4583.294} C_VEL
LIN {X 0,Y 72.54,Z 475.669,A -85,B 0,C 180,E1 4577.356,E2 4577.356} C_VEL
LIN {X 0,Y 69.181,Z 474.232,A -85,B 0,C 180,E1 4566.876,E2 4566.876} C_VEL
LIN {X 0,Y 68.783,Z 472.397,A -85,B 0,C 180,E1 4558.646,E2 4558.646} C_VEL
LIN {X 0,Y 69.825,Z 471.437,A -85,B 0,C 180,E1 4555.15,E2 4555.15} C_VEL
LIN {X 0,Y 76.677,Z 467.048,A -85,B 0,C 180,E1 4544.186,E2 4544.186} C_VEL
LIN {X 0,Y 85.189,Z 461.107,A -85,B 0,C 180,E1 4535.929,E2 4535.929} C_VEL
LIN {X 0,Y 94.445,Z 453.79,A -85,B 0,C 180,E1 4529.771,E2 4529.771} C_VEL
LIN {X 0,Y 104.639,Z 444.342,A -85,B 0,C 180,E1 4524.815,E2 4524.815} C_VEL
LIN {X 0,Y 114.663,Z 433.131,A -85,B 0,C 180,E1 4521.1,E2 4521.1} C_VEL
LIN {X 0,Y 123.351,Z 421.202,A -85,B 0,C 180,E1 4518.504,E2 4518.504} C_VEL
LIN {X 0,Y 130.473,Z 409.133,A -85,B 0,C 180,E1 4516.696,E2 4516.696} C_VEL
LIN {X 0,Y 136.971,Z 394.903,A -85,B 0,C 180,E1 4515.235,E2 4515.235} C_VEL
LIN {X 0,Y 141.914,Z 379.697,A -85,B 0,C 180,E1 4514.222,E2 4514.222} C_VEL
LIN {X 0,Y 144.914,Z 364.971,A -85,B 0,C 180,E1 4513.61,E2 4513.61} C_VEL
LIN {X 0,Y 157.942,Z 249.776,A -85,B 0,C 180,E1 4510.253,E2 4510.253} C_VEL
LIN {X 0,Y 159.382,Z 244.239,A -85,B 0,C 180,E1 4509.986,E2 4509.986} C_VEL
LIN {X 0,Y 163.022,Z 233.362,A -85,B 0,C 180,E1 4509.442,E2 4509.442} C_VEL
LIN {X 0,Y 162.436,Z 231.823,A -85,B 0,C 180,E1 4506.006,E2 4506.006} C_VEL
LIN {X 0,Y 161.121,Z 234.064,A -85,B 0,C 180,E1 4498.933,E2 4498.933} C_VEL
LIN {X 0,Y 160.754,Z 237.291,A -85,B 0,C 180,E1 4494.646,E2 4494.646} C_VEL
LIN {X 0,Y 160.536,Z 241.691,A -85,B 0,C 180,E1 4490.77,E2 4490.77} C_VEL
LIN {X 0,Y 161.639,Z 246.61,A -85,B 0,C 180,E1 4488.059,E2 4488.059} C_VEL
LIN {X 0,Y 161.352,Z 251.111,A -85,B 0,C 180,E1 4487.659,E2 4487.659} C_VEL
LIN {X 0,Y 153.4,Z 324.613,A -85,B 0,C 180,E1 4485.76,E2 4485.76} C_VEL
LIN {X 0,Y 149.969,Z 358.126,A -85,B 0,C 180,E1 4484.302,E2 4484.302} C_VEL
LIN {X 0,Y 146.721,Z 373.401,A -85,B 0,C 180,E1 4483.215,E2 4483.215} C_VEL
LIN {X 0,Y 141.634,Z 388.332,A -85,B 0,C 180,E1 4481.7,E2 4481.7} C_VEL
LIN {X 0,Y 135.282,Z 401.633,A -85,B 0,C 180,E1 4479.813,E2 4479.813} C_VEL
LIN {X 0,Y 128.028,Z 413.377,A -85,B 0,C 180,E1 4477.499,E2 4477.499} C_VEL
LIN {X 0,Y 119.627,Z 424.241,A -85,B 0,C 180,E1 4474.502,E2 4474.502} C_VEL
LIN {X 0,Y 110.194,Z 434.024,A -85,B 0,C 180,E1 4470.573,E2 4470.573} C_VEL
LIN {X 0,Y 100.54,Z 442.086,A -85,B 0,C 180,E1 4465.622,E2 4465.622} C_VEL
LIN {X 0,Y 91.664,Z 448.1,A -85,B 0,C 180,E1 4459.769,E2 4459.769} C_VEL
LIN {X 0,Y 83.255,Z 452.666,A -85,B 0,C 180,E1 4452.255,E2 4452.255} C_VEL
LIN {X 0,Y 75.549,Z 455.712,A -85,B 0,C 180,E1 4441.956,E2 4441.956} C_VEL
LIN {X 0,Y 70.436,Z 456.647,A -85,B 0,C 180,E1 4429.912,E2 4429.912} C_VEL
LIN {X 0,Y 68.387,Z 455.653,A -85,B 0,C 180,E1 4417.555,E2 4417.555} C_VEL
LIN {X 0,Y 69.011,Z 453.128,A -85,B 0,C 180,E1 4405.839,E2 4405.839} C_VEL
LIN {X 0,Y 72.3,Z 448.58,A -85,B 0,C 180,E1 4393.938,E2 4393.938} C_VEL
LIN {X 0,Y 72.971,Z 447.612,A -85,B 0,C 180,E1 4392.037,E2 4392.037} C_VEL
LIN {X 0,Y 69.068,Z 445.655,A -85,B 0,C 180,E1 4383.841,E2 4383.841} C_VEL
LIN {X 0,Y 67.965,Z 451.978,A -85,B 0,C 180,E1 4369.654,E2 4369.654} C_VEL
LIN {X 0,Y 70.606,Z 456.484,A -85,B 0,C 180,E1 4355.495,E2 4355.495} C_VEL
LIN {X 0,Y 76.966,Z 459.191,A -85,B 0,C 180,E1 4342.716,E2 4342.716} C_VEL
LIN {X 0,Y 86.636,Z 460.024,A -85,B 0,C 180,E1 4331.991,E2 4331.991} C_VEL
LIN {X 0,Y 98.216,Z 459.077,A -85,B 0,C 180,E1 4323.871,E2 4323.871} C_VEL
LIN {X 0,Y 111.082,Z 456.408,A -85,B 0,C 180,E1 4317.669,E2 4317.669} C_VEL
LIN {X 0,Y 125.423,Z 451.742,A -85,B 0,C 180,E1 4312.673,E2 4312.673} C_VEL
LIN {X 0,Y 139.939,Z 445.324,A -85,B 0,C 180,E1 4308.878,E2 4308.878} C_VEL
LIN {X 0,Y 151.152,Z 439.127,A -85,B 0,C 180,E1 4306.514,E2 4306.514} C_VEL
LIN {X 0,Y 136.288,Z 448.507,A -85,B 0,C 180,E1 4303.967,E2 4303.967} C_VEL
LIN {X 0,Y 120.121,Z 456.948,A -85,B 0,C 180,E1 4300.158,E2 4300.158} C_VEL
LIN {X 0,Y 104.823,Z 463.397,A -85,B 0,C 180,E1 4294.988,E2 4294.988} C_VEL
LIN {X 0,Y 90.153,Z 468.34,A -85,B 0,C 180,E1 4287.454,E2 4287.454} C_VEL
LIN {X 0,Y 77.898,Z 471.538,A -85,B 0,C 180,E1 4277.029,E2 4277.029} C_VEL
LIN {X 0,Y 69.058,Z 473.094,A -85,B 0,C 180,E1 4262.399,E2 4262.399} C_VEL
LIN {X 0,Y 66.01,Z 472.721,A -85,B 0,C 180,E1 4244.928,E2 4244.928} C_VEL
LIN {X 0,Y 66.439,Z 472.192,A -85,B 0,C 180,E1 4238.662,E2 4238.662} C_VEL
LIN {X 0,Y 67.629,Z 474.169,A -85,B 0,C 180,E1 4230.006,E2 4230.006} C_VEL
LIN {X 0,Y 65.547,Z 474.601,A -85,B 0,C 180,E1 4215.881,E2 4215.881} C_VEL
LIN {X 0,Y 67.192,Z 473.131,A -85,B 0,C 180,E1 4202.537,E2 4202.537} C_VEL
LIN {X 0,Y 69.825,Z 471.437,A -85,B 0,C 180,E1 4195.15,E2 4195.15} C_VEL
LIN {X 0,Y 71.863,Z 469.524,A -85,B 0,C 180,E1 4189.281,E2 4189.281} C_VEL
LIN {X 0,Y 75.698,Z 464.3,A -85,B 0,C 180,E1 4177.225,E2 4177.225} C_VEL
LIN {X 0,Y 79.698,Z 460.838,A -85,B 0,C 180,E1 4171.955,E2 4171.955} C_VEL
LIN {X 0,Y 81.059,Z 459.884,A -85,B 0,C 180,E1 4170.899,E2 4170.899} C_VEL
LIN {X 0,Y 91.461,Z 452.266,A -85,B 0,C 180,E1 4164.871,E2 4164.871} C_VEL
LIN {X 0,Y 101.481,Z 443.548,A -85,B 0,C 180,E1 4160.624,E2 4160.624} C_VEL
LIN {X 0,Y 111.362,Z 433.159,A -85,B 0,C 180,E1 4157.39,E2 4157.39} C_VEL
LIN {X 0,Y 120.109,Z 421.982,A -85,B 0,C 180,E1 4155.078,E2 4155.078} C_VEL
LIN {X 0,Y 128.384,Z 408.763,A -85,B 0,C 180,E1 4153.238,E2 4153.238} C_VEL
LIN {X 0,Y 134.907,Z 395.158,A -85,B 0,C 180,E1 4151.974,E2 4151.974} C_VEL
LIN {X 0,Y 139.923,Z 380.881,A -85,B 0,C 180,E1 4151.094,E2 4151.094} C_VEL
LIN {X 0,Y 143.372,Z 365.817,A -85,B 0,C 180,E1 4150.503,E2 4150.503} C_VEL
LIN {X 0,Y 156.933,Z 250.476,A -85,B 0,C 180,E1 4147.376,E2 4147.376} C_VEL
LIN {X 0,Y 157.708,Z 245.862,A -85,B 0,C 180,E1 4147.191,E2 4147.191} C_VEL
LIN {X 0,Y 159.799,Z 239.762,A -85,B 0,C 180,E1 4146.917,E2 4146.917} C_VEL
LIN {X 0,Y 159.609,Z 239.454,A -85,B 0,C 180,E1 4145.752,E2 4145.752} C_VEL
LIN {X 0,Y 158.317,Z 241.578,A -85,B 0,C 180,E1 4139.276,E2 4139.276} C_VEL
LIN {X 0,Y 158.003,Z 243.957,A -85,B 0,C 180,E1 4136.008,E2 4136.008} C_VEL
LIN {X 0,Y 159.007,Z 248.826,A -85,B 0,C 180,E1 4131.957,E2 4131.957} C_VEL
LIN {X 0,Y 159.482,Z 251.577,A -85,B 0,C 180,E1 4130.434,E2 4130.434} C_VEL
LIN {X 0,Y 151.269,Z 325.118,A -85,B 0,C 180,E1 4128.654,E2 4128.654} C_VEL
LIN {X 0,Y 147.595,Z 359.192,A -85,B 0,C 180,E1 4127.219,E2 4127.219} C_VEL
LIN {X 0,Y 144.373,Z 373.893,A -85,B 0,C 180,E1 4126.224,E2 4126.224} C_VEL
LIN {X 0,Y 139.754,Z 387.374,A -85,B 0,C 180,E1 4124.966,E2 4124.966} C_VEL
LIN {X 0,Y 134.04,Z 399.678,A -85,B 0,C 180,E1 4123.428,E2 4123.428} C_VEL
LIN {X 0,Y 126.205,Z 412.527,A -85,B 0,C 180,E1 4121.202,E2 4121.202} C_VEL
LIN {X 0,Y 117.243,Z 423.977,A -85,B 0,C 180,E1 4118.354,E2 4118.354} C_VEL
LIN {X 0,Y 108.11,Z 433.313,A -85,B 0,C 180,E1 4114.995,E2 4114.995} C_VEL
LIN {X 0,Y 98.555,Z 441.285,A -85,B 0,C 180,E1 4110.738,E2 4110.738} C_VEL
LIN {X 0,Y 88.123,Z 448.233,A -85,B 0,C 180,E1 4104.769,E2 4104.769} C_VEL
LIN {X 0,Y 78.746,Z 453.087,A -85,B 0,C 180,E1 4097.42,E2 4097.42} C_VEL
LIN {X 0,Y 70.825,Z 456.17,A -85,B 0,C 180,E1 4088.392,E2 4088.392} C_VEL
LIN {X 0,Y 64.5,Z 457.657,A -85,B 0,C 180,E1 4076.707,E2 4076.707} C_VEL
LIN {X 0,Y 60.857,Z 457.233,A -85,B 0,C 180,E1 4062.325,E2 4062.325} C_VEL
LIN {X 0,Y 60.728,Z 454.981,A -85,B 0,C 180,E1 4048.106,E2 4048.106} C_VEL
LIN {X 0,Y 63.468,Z 451.22,A -85,B 0,C 180,E1 4035.394,E2 4035.394} C_VEL
LIN {X 0,Y 64.669,Z 449.838,A -85,B 0,C 180,E1 4031.981,E2 4031.981} C_VEL
LIN {X 0,Y 60.597,Z 447.806,A -85,B 0,C 180,E1 4021.674,E2 4021.674} C_VEL
LIN {X 0,Y 60.51,Z 454.341,A -85,B 0,C 180,E1 4003.951,E2 4003.951} C_VEL
LIN {X 0,Y 64.453,Z 458.206,A -85,B 0,C 180,E1 3989.677,E2 3989.677} C_VEL
LIN {X 0,Y 72.843,Z 460.667,A -85,B 0,C 180,E1 3976.071,E2 3976.071} C_VEL
LIN {X 0,Y 84.399,Z 461.254,A -85,B 0,C 180,E1 3965.613,E2 3965.613} C_VEL
LIN {X 0,Y 98.062,Z 459.854,A -85,B 0,C 180,E1 3957.838,E2 3957.838} C_VEL
LIN {X 0,Y 113.072,Z 456.503,A -85,B 0,C 180,E1 3952.066,E2 3952.066} C_VEL
LIN {X 0,Y 128.314,Z 451.333,A -85,B 0,C 180,E1 3947.856,E2 3947.856} C_VEL
LIN {X 0,Y 132.171,Z 449.74,A -85,B 0,C 180,E1 3946.912,E2 3946.912} C_VEL
LIN {X 0,Y 115.796,Z 457.455,A -85,B 0,C 180,E1 3943.435,E2 3943.435} C_VEL
LIN {X 0,Y 99.071,Z 463.743,A -85,B 0,C 180,E1 3938.211,E2 3938.211} C_VEL
LIN {X 0,Y 83.721,Z 468.12,A -85,B 0,C 180,E1 3930.679,E2 3930.679} C_VEL
LIN {X 0,Y 70.119,Z 470.865,A -85,B 0,C 180,E1 3919.099,E2 3919.099} C_VEL
LIN {X 0,Y 60.929,Z 471.799,A -85,B 0,C 180,E1 3902.796,E2 3902.796} C_VEL
LIN {X 0,Y 58.252,Z 470.863,A -85,B 0,C 180,E1 3882.901,E2 3882.901} C_VEL
LIN {X 0,Y 58.393,Z 470.954,A -85,B 0,C 180,E1 3879.867,E2 3879.867} C_VEL
LIN {X 0,Y 59.512,Z 472.994,A -85,B 0,C 180,E1 3870.007,E2 3870.007} C_VEL
LIN {X 0,Y 57.617,Z 473.481,A -85,B 0,C 180,E1 3854.92,E2 3854.92} C_VEL
LIN {X 0,Y 59.725,Z 472.197,A -85,B 0,C 180,E1 3839.861,E2 3839.861} C_VEL
LIN {X 0,Y 65.598,Z 469.14,A -85,B 0,C 180,E1 3826.704,E2 3826.704} C_VEL
LIN {X 0,Y 75.034,Z 463.769,A -85,B 0,C 180,E1 3815.636,E2 3815.636} C_VEL
LIN {X 0,Y 81.059,Z 459.884,A -85,B 0,C 180,E1 3810.899,E2 3810.899} C_VEL
LIN {X 0,Y 85.501,Z 456.441,A -85,B 0,C 180,E1 3807.201,E2 3807.201} C_VEL
LIN {X 0,Y 92.426,Z 449.424,A -85,B 0,C 180,E1 3800.3,E2 3800.3} C_VEL
LIN {X 0,Y 97.283,Z 444.403,A -85,B 0,C 180,E1 3796.956,E2 3796.956} C_VEL
LIN {X 0,Y 100.123,Z 441.637,A -85,B 0,C 180,E1 3795.801,E2 3795.801} C_VEL
LIN {X 0,Y 110.778,Z 430.721,A -85,B 0,C 180,E1 3792.915,E2 3792.915} C_VEL
LIN {X 0,Y 120.137,Z 418.763,A -85,B 0,C 180,E1 3790.891,E2 3790.891} C_VEL
LIN {X 0,Y 127.728,Z 406.651,A -85,B 0,C 180,E1 3789.512,E2 3789.512} C_VEL
LIN {X 0,Y 134.43,Z 392.794,A -85,B 0,C 180,E1 3788.448,E2 3788.448} C_VEL
LIN {X 0,Y 139.67,Z 377.571,A -85,B 0,C 180,E1 3787.708,E2 3787.708} C_VEL
LIN {X 0,Y 142.883,Z 362.613,A -85,B 0,C 180,E1 3787.237,E2 3787.237} C_VEL
LIN {X 0,Y 156.359,Z 250.89,A -85,B 0,C 180,E1 3784.458,E2 3784.458} C_VEL
LIN {X 0,Y 156.753,Z 247.566,A -85,B 0,C 180,E1 3784.297,E2 3784.297} C_VEL
LIN {X 0,Y 156.567,Z 249.26,A -85,B 0,C 180,E1 3779.816,E2 3779.816} C_VEL
LIN {X 0,Y 156.934,Z 252.193,A -85,B 0,C 180,E1 3776.163,E2 3776.163} C_VEL
LIN {X 0,Y 157.521,Z 256.098,A -85,B 0,C 180,E1 3773.188,E2 3773.188} C_VEL
LIN {X 0,Y 149.497,Z 325.952,A -85,B 0,C 180,E1 3771.613,E2 3771.613} C_VEL
LIN {X 0,Y 145.588,Z 360.412,A -85,B 0,C 180,E1 3770.214,E2 3770.214} C_VEL
LIN {X 0,Y 142.209,Z 375.185,A -85,B 0,C 180,E1 3769.265,E2 3769.265} C_VEL
LIN {X 0,Y 136.974,Z 389.705,A -85,B 0,C 180,E1 3767.981,E2 3767.981} C_VEL
LIN {X 0,Y 130.611,Z 402.452,A -85,B 0,C 180,E1 3766.444,E2 3766.444} C_VEL
LIN {X 0,Y 123.404,Z 413.707,A -85,B 0,C 180,E1 3764.6,E2 3764.6} C_VEL
LIN {X 0,Y 114.089,Z 425.141,A -85,B 0,C 180,E1 3761.952,E2 3761.952} C_VEL
LIN {X 0,Y 104.12,Z 434.834,A -85,B 0,C 180,E1 3758.654,E2 3758.654} C_VEL
LIN {X 0,Y 94.076,Z 442.7,A -85,B 0,C 180,E1 3754.595,E2 3754.595} C_VEL
LIN {X 0,Y 82.996,Z 449.572,A -85,B 0,C 180,E1 3748.785,E2 3748.785} C_VEL
LIN {X 0,Y 72.212,Z 454.634,A -85,B 0,C 180,E1 3740.829,E2 3740.829} C_VEL
LIN {X 0,Y 62.972,Z 457.677,A -85,B 0,C 180,E1 3730.344,E2 3730.344} C_VEL
LIN {X 0,Y 56.36,Z 458.803,A -85,B 0,C 180,E1 3717.459,E2 3717.459} C_VEL
LIN {X 0,Y 52.839,Z 458.182,A -85,B 0,C 180,E1 3702.005,E2 3702.005} C_VEL
LIN {X 0,Y 53.031,Z 455.75,A -85,B 0,C 180,E1 3685.667,E2 3685.667} C_VEL
LIN {X 0,Y 56.327,Z 451.943,A -85,B 0,C 180,E1 3671.894,E2 3671.894} C_VEL
LIN {X 0,Y 52.182,Z 449.921,A -85,B 0,C 180,E1 3658.515,E2 3658.515} C_VEL
LIN {X 0,Y 53.162,Z 455.851,A -85,B 0,C 180,E1 3639.534,E2 3639.534} C_VEL
LIN {X 0,Y 58.937,Z 459.766,A -85,B 0,C 180,E1 3622.969,E2 3622.969} C_VEL
LIN {X 0,Y 69.425,Z 462.098,A -85,B 0,C 180,E1 3609.117,E2 3609.117} C_VEL
LIN {X 0,Y 81.996,Z 462.465,A -85,B 0,C 180,E1 3599.718,E2 3599.718} C_VEL
LIN {X 0,Y 96.775,Z 460.94,A -85,B 0,C 180,E1 3592.706,E2 3592.706} C_VEL
LIN {X 0,Y 112.597,Z 457.521,A -85,B 0,C 180,E1 3587.647,E2 3587.647} C_VEL
LIN {X 0,Y 113.67,Z 457.235,A -85,B 0,C 180,E1 3587.365,E2 3587.365} C_VEL
LIN {X 0,Y 96.338,Z 463.12,A -85,B 0,C 180,E1 3582.727,E2 3582.727} C_VEL
LIN {X 0,Y 79.214,Z 467.395,A -85,B 0,C 180,E1 3575.351,E2 3575.351} C_VEL
LIN {X 0,Y 64.31,Z 469.836,A -85,B 0,C 180,E1 3563.788,E2 3563.788} C_VEL
LIN {X 0,Y 53.868,Z 470.374,A -85,B 0,C 180,E1 3546.448,E2 3546.448} C_VEL
LIN {X 0,Y 50.394,Z 469.278,A -85,B 0,C 180,E1 3523.549,E2 3523.549} C_VEL
LIN {X 0,Y 51.384,Z 471.809,A -85,B 0,C 180,E1 3510.008,E2 3510.008} C_VEL
LIN {X 0,Y 49.738,Z 472.339,A -85,B 0,C 180,E1 3492.46,E2 3492.46} C_VEL
LIN {X 0,Y 52.765,Z 471.109,A -85,B 0,C 180,E1 3475.367,E2 3475.367} C_VEL
LIN {X 0,Y 60.457,Z 467.827,A -85,B 0,C 180,E1 3460.481,E2 3460.481} C_VEL
LIN {X 0,Y 70.551,Z 462.782,A -85,B 0,C 180,E1 3450.189,E2 3450.189} C_VEL
LIN {X 0,Y 81.564,Z 456.135,A -85,B 0,C 180,E1 3443.179,E2 3443.179} C_VEL
LIN {X 0,Y 92.668,Z 448.034,A -85,B 0,C 180,E1 3438.306,E2 3438.306} C_VEL
LIN {X 0,Y 100.123,Z 441.637,A -85,B 0,C 180,E1 3435.801,E2 3435.801} C_VEL
LIN {X 0,Y 104.886,Z 436.673,A -85,B 0,C 180,E1 3433.802,E2 3433.802} C_VEL
LIN {X 0,Y 114.084,Z 424.849,A -85,B 0,C 180,E1 3428.674,E2 3428.674} C_VEL
LIN {X 0,Y 118.275,Z 419.062,A -85,B 0,C 180,E1 3427.192,E2 3427.192} C_VEL
LIN {X 0,Y 119.544,Z 417.288,A -85,B 0,C 180,E1 3426.945,E2 3426.945} C_VEL
LIN {X 0,Y 127.621,Z 404.524,A -85,B 0,C 180,E1 3425.778,E2 3425.778} C_VEL
LIN {X 0,Y 133.977,Z 391.53,A -85,B 0,C 180,E1 3424.981,E2 3424.981} C_VEL
LIN {X 0,Y 139.317,Z 376.25,A -85,B 0,C 180,E1 3424.392,E2 3424.392} C_VEL
LIN {X 0,Y 142.56,Z 361.334,A -85,B 0,C 180,E1 3424.005,E2 3424.005} C_VEL
LIN {X 0,Y 155.556,Z 256.431,A -85,B 0,C 180,E1 3421.65,E2 3421.65} C_VEL
LIN {X 0,Y 155.684,Z 259.021,A -85,B 0,C 180,E1 3417.791,E2 3417.791} C_VEL
LIN {X 0,Y 155.879,Z 261.07,A -85,B 0,C 180,E1 3415.998,E2 3415.998} C_VEL
LIN {X 0,Y 148.119,Z 326.953,A -85,B 0,C 180,E1 3414.629,E2 3414.629} C_VEL
LIN {X 0,Y 144.018,Z 361.479,A -85,B 0,C 180,E1 3413.291,E2 3413.291} C_VEL
LIN {X 0,Y 140.457,Z 376.47,A -85,B 0,C 180,E1 3412.39,E2 3412.39} C_VEL
LIN {X 0,Y 135.057,Z 390.935,A -85,B 0,C 180,E1 3411.213,E2 3411.213} C_VEL
LIN {X 0,Y 128.497,Z 403.65,A -85,B 0,C 180,E1 3409.816,E2 3409.816} C_VEL
LIN {X 0,Y 120.594,Z 415.492,A -85,B 0,C 180,E1 3408.034,E2 3408.034} C_VEL
LIN {X 0,Y 111.409,Z 426.305,A -85,B 0,C 180,E1 3405.738,E2 3405.738} C_VEL
LIN {X 0,Y 101.478,Z 435.61,A -85,B 0,C 180,E1 3402.871,E2 3402.871} C_VEL
LIN {X 0,Y 90.929,Z 443.559,A -85,B 0,C 180,E1 3399.158,E2 3399.158} C_VEL
LIN {X 0,Y 79.144,Z 450.49,A -85,B 0,C 180,E1 3393.749,E2 3393.749} C_VEL
LIN {X 0,Y 68.183,Z 455.324,A -85,B 0,C 180,E1 3386.694,E2 3386.694} C_VEL
LIN {X 0,Y 58.49,Z 458.387,A -85,B 0,C 180,E1 3377.301,E2 3377.301} C_VEL
LIN {X 0,Y 50.285,Z 459.858,A -85,B 0,C 180,E1 3363.82,E2 3363.82} C_VEL
LIN {X 0,Y 45.235,Z 459.414,A -85,B 0,C 180,E1 3345.371,E2 3345.371} C_VEL
LIN {X 0,Y 44.966,Z 457.139,A -85,B 0,C 180,E1 3326.165,E2 3326.165} C_VEL
LIN {X 0,Y 47.91,Z 454.006,A -85,B 0,C 180,E1 3311.748,E2 3311.748} C_VEL
LIN {X 0,Y 43.956,Z 452,A -85,B 0,C 180,E1 3294.174,E2 3294.174} C_VEL
LIN {X 0,Y 46.542,Z 457.572,A -85,B 0,C 180,E1 3272.488,E2 3272.488} C_VEL
LIN {X 0,Y 54.74,Z 461.435,A -85,B 0,C 180,E1 3254.487,E2 3254.487} C_VEL
LIN {X 0,Y 67.025,Z 463.485,A -85,B 0,C 180,E1 3241.652,E2 3241.652} C_VEL
LIN {X 0,Y 81.727,Z 463.588,A -85,B 0,C 180,E1 3232.974,E2 3232.974} C_VEL
LIN {X 0,Y 95.169,Z 462.244,A -85,B 0,C 180,E1 3227.725,E2 3227.725} C_VEL
LIN {X 0,Y 77.908,Z 466.165,A -85,B 0,C 180,E1 3221.765,E2 3221.765} C_VEL
LIN {X 0,Y 61.417,Z 468.487,A -85,B 0,C 180,E1 3211.548,E2 3211.548} C_VEL
LIN {X 0,Y 48.524,Z 468.961,A -85,B 0,C 180,E1 3194.485,E2 3194.485} C_VEL
LIN {X 0,Y 42.597,Z 467.723,A -85,B 0,C 180,E1 3167.777,E2 3167.777} C_VEL
LIN {X 0,Y 43.247,Z 470.621,A -85,B 0,C 180,E1 3150.01,E2 3150.01} C_VEL
LIN {X 0,Y 41.982,Z 471.196,A -85,B 0,C 180,E1 3129.08,E2 3129.08} C_VEL
LIN {X 0,Y 46.229,Z 470.021,A -85,B 0,C 180,E1 3109.559,E2 3109.559} C_VEL
LIN {X 0,Y 55.48,Z 466.784,A -85,B 0,C 180,E1 3093.962,E2 3093.962} C_VEL
LIN {X 0,Y 67.605,Z 461.407,A -85,B 0,C 180,E1 3083.532,E2 3083.532} C_VEL
LIN {X 0,Y 80.466,Z 454.137,A -85,B 0,C 180,E1 3076.926,E2 3076.926} C_VEL
LIN {X 0,Y 92.278,Z 445.761,A -85,B 0,C 180,E1 3072.819,E2 3072.819} C_VEL
LIN {X 0,Y 103.532,Z 435.922,A -85,B 0,C 180,E1 3069.944,E2 3069.944} C_VEL
LIN {X 0,Y 114.049,Z 424.497,A -85,B 0,C 180,E1 3067.87,E2 3067.87} C_VEL
LIN {X 0,Y 119.544,Z 417.288,A -85,B 0,C 180,E1 3066.945,E2 3066.945} C_VEL
LIN {X 0,Y 123.663,Z 411.109,A -85,B 0,C 180,E1 3065.849,E2 3065.849} C_VEL
LIN {X 0,Y 130.324,Z 398.616,A -85,B 0,C 180,E1 3062.821,E2 3062.821} C_VEL
LIN {X 0,Y 133.746,Z 390.916,A -85,B 0,C 180,E1 3061.623,E2 3061.623} C_VEL
LIN {X 0,Y 134.991,Z 387.852,A -85,B 0,C 180,E1 3061.434,E2 3061.434} C_VEL
LIN {X 0,Y 139.82,Z 373.535,A -85,B 0,C 180,E1 3061.036,E2 3061.036} C_VEL
LIN {X 0,Y 143.089,Z 357.547,A -85,B 0,C 180,E1 3060.683,E2 3060.683} C_VEL
LIN {X 0,Y 154.575,Z 266.375,A -85,B 0,C 180,E1 3058.887,E2 3058.887} C_VEL
LIN {X 0,Y 146.91,Z 330.096,A -85,B 0,C 180,E1 3057.632,E2 3057.632} C_VEL
LIN {X 0,Y 142.83,Z 362.762,A -85,B 0,C 180,E1 3056.417,E2 3056.417} C_VEL
LIN {X 0,Y 139.374,Z 376.944,A -85,B 0,C 180,E1 3055.636,E2 3055.636} C_VEL
LIN {X 0,Y 134.209,Z 390.739,A -85,B 0,C 180,E1 3054.646,E2 3054.646} C_VEL
LIN {X 0,Y 127.803,Z 403.271,A -85,B 0,C 180,E1 3053.465,E2 3053.465} C_VEL
LIN {X 0,Y 119.109,Z 416.17,A -85,B 0,C 180,E1 3051.794,E2 3051.794} C_VEL
LIN {X 0,Y 108.768,Z 427.957,A -85,B 0,C 180,E1 3049.585,E2 3049.585} C_VEL
LIN {X 0,Y 97.561,Z 437.878,A -85,B 0,C 180,E1 3046.785,E2 3046.785} C_VEL
LIN {X 0,Y 86.587,Z 445.526,A -85,B 0,C 180,E1 3043.403,E2 3043.403} C_VEL
LIN {X 0,Y 75.075,Z 451.826,A -85,B 0,C 180,E1 3038.774,E2 3038.774} C_VEL
LIN {X 0,Y 62.527,Z 456.871,A -85,B 0,C 180,E1 3031.565,E2 3031.565} C_VEL
LIN {X 0,Y 51.287,Z 459.862,A -85,B 0,C 180,E1 3021.229,E2 3021.229} C_VEL
LIN {X 0,Y 42.33,Z 461,A -85,B 0,C 180,E1 3006.18,E2 3006.18} C_VEL
LIN {X 0,Y 37.211,Z 460.356,A -85,B 0,C 180,E1 2985.574,E2 2985.574} C_VEL
LIN {X 0,Y 37.387,Z 457.908,A -85,B 0,C 180,E1 2962.304,E2 2962.304} C_VEL
LIN {X 0,Y 39.424,Z 455.965,A -85,B 0,C 180,E1 2951.397,E2 2951.397} C_VEL
LIN {X 0,Y 36.072,Z 454.031,A -85,B 0,C 180,E1 2927.749,E2 2927.749} C_VEL
LIN {X 0,Y 41.134,Z 459.454,A -85,B 0,C 180,E1 2902.504,E2 2902.504} C_VEL
LIN {X 0,Y 52.166,Z 463.119,A -85,B 0,C 180,E1 2884.577,E2 2884.577} C_VEL
LIN {X 0,Y 66.432,Z 464.841,A -85,B 0,C 180,E1 2873.44,E2 2873.44} C_VEL
LIN {X 0,Y 77.258,Z 465.015,A -85,B 0,C 180,E1 2868.182,E2 2868.182} C_VEL
LIN {X 0,Y 59.656,Z 467.134,A -85,B 0,C 180,E1 2859.834,E2 2859.834} C_VEL
LIN {X 0,Y 44.172,Z 467.522,A -85,B 0,C 180,E1 2843.951,E2 2843.951} C_VEL
LIN {X 0,Y 35.464,Z 466.162,A -85,B 0,C 180,E1 2816.827,E2 2816.827} C_VEL
LIN {X 0,Y 35.085,Z 466.197,A -85,B 0,C 180,E1 2813.527,E2 2813.527} C_VEL
LIN {X 0,Y 35.1,Z 469.432,A -85,B 0,C 180,E1 2790.012,E2 2790.012} C_VEL
LIN {X 0,Y 34.442,Z 470.053,A -85,B 0,C 180,E1 2764.143,E2 2764.143} C_VEL
LIN {X 0,Y 40.318,Z 468.932,A -85,B 0,C 180,E1 2741.946,E2 2741.946} C_VEL
LIN {X 0,Y 51.307,Z 465.749,A -85,B 0,C 180,E1 2726.328,E2 2726.328} C_VEL
LIN {X 0,Y 63.912,Z 460.794,A -85,B 0,C 180,E1 2717.29,E2 2717.29} C_VEL
LIN {X 0,Y 76.602,Z 454.308,A -85,B 0,C 180,E1 2711.809,E2 2711.809} C_VEL
LIN {X 0,Y 88.895,Z 446.371,A -85,B 0,C 180,E1 2708.233,E2 2708.233} C_VEL
LIN {X 0,Y 101.464,Z 436.114,A -85,B 0,C 180,E1 2705.621,E2 2705.621} C_VEL
LIN {X 0,Y 112.731,Z 424.441,A -85,B 0,C 180,E1 2703.867,E2 2703.867} C_VEL
LIN {X 0,Y 121.614,Z 412.83,A -85,B 0,C 180,E1 2702.757,E2 2702.757} C_VEL
LIN {X 0,Y 129.549,Z 399.669,A -85,B 0,C 180,E1 2701.929,E2 2701.929} C_VEL
LIN {X 0,Y 134.991,Z 387.852,A -85,B 0,C 180,E1 2701.434,E2 2701.434} C_VEL
LIN {X 0,Y 134.779,Z 388.347,A -85,B 0,C 180,E1 2701.118,E2 2701.118} C_VEL
LIN {X 0,Y 133.149,Z 392.086,A -85,B 0,C 180,E1 2700.539,E2 2700.539} C_VEL
LIN {X 0,Y 126.336,Z 404.994,A -85,B 0,C 180,E1 2699.539,E2 2699.539} C_VEL
LIN {X 0,Y 119.974,Z 414.487,A -85,B 0,C 180,E1 2699.158,E2 2699.158} C_VEL
LIN {X 0,Y 117.232,Z 418.096,A -85,B 0,C 180,E1 2699.285,E2 2699.285} C_VEL
LIN {X 0,Y 106.477,Z 430.176,A -85,B 0,C 180,E1 2700.346,E2 2700.346} C_VEL
LIN {X 0,Y 95.026,Z 440.345,A -85,B 0,C 180,E1 2701.827,E2 2701.827} C_VEL
LIN {X 0,Y 83.171,Z 448.801,A -85,B 0,C 180,E1 2703.893,E2 2703.893} C_VEL
LIN {X 0,Y 69.014,Z 456.675,A -85,B 0,C 180,E1 2707.49,E2 2707.49} C_VEL
LIN {X 0,Y 54.497,Z 462.679,A -85,B 0,C 180,E1 2713.535,E2 2713.535} C_VEL
LIN {X 0,Y 41.452,Z 466.506,A -85,B 0,C 180,E1 2723.594,E2 2723.594} C_VEL
LIN {X 0,Y 30.865,Z 468.548,A -85,B 0,C 180,E1 2741.857,E2 2741.857} C_VEL
LIN {X 0,Y 25.965,Z 468.792,A -85,B 0,C 180,E1 2774.38,E2 2774.38} C_VEL
LIN {X 0,Y 27.002,Z 468.15,A -85,B 0,C 180,E1 2791.374,E2 2791.374} C_VEL
LIN {X 0,Y 28.484,Z 464.432,A -85,B 0,C 180,E1 2824.187,E2 2824.187} C_VEL
LIN {X 0,Y 40.146,Z 466.05,A -85,B 0,C 180,E1 2853.739,E2 2853.739} C_VEL
LIN {X 0,Y 57.354,Z 465.889,A -85,B 0,C 180,E1 2867.519,E2 2867.519} C_VEL
LIN {X 0,Y 59.707,Z 465.739,A -85,B 0,C 180,E1 2868.71,E2 2868.71} C_VEL
LIN {X 0,Y 44.003,Z 463.275,A -85,B 0,C 180,E1 2880.604,E2 2880.604} C_VEL
LIN {X 0,Y 32.946,Z 459.36,A -85,B 0,C 180,E1 2899.775,E2 2899.775} C_VEL
LIN {X 0,Y 28.648,Z 455.911,A -85,B 0,C 180,E1 2919.817,E2 2919.817} C_VEL
LIN {X 0,Y 30.962,Z 457.936,A -85,B 0,C 180,E1 2951.625,E2 2951.625} C_VEL
LIN {X 0,Y 28.778,Z 460.905,A -85,B 0,C 180,E1 2979.989,E2 2979.989} C_VEL
LIN {X 0,Y 33.943,Z 462.123,A -85,B 0,C 180,E1 3008.196,E2 3008.196} C_VEL
LIN {X 0,Y 43.646,Z 461.395,A -85,B 0,C 180,E1 3025.539,E2 3025.539} C_VEL
LIN {X 0,Y 54.849,Z 459.079,A -85,B 0,C 180,E1 3035.688,E2 3035.688} C_VEL
LIN {X 0,Y 68.009,Z 454.693,A -85,B 0,C 180,E1 3042.84,E2 3042.84} C_VEL
LIN {X 0,Y 80.895,Z 448.556,A -85,B 0,C 180,E1 3047.506,E2 3047.506} C_VEL
LIN {X 0,Y 93.179,Z 440.774,A -85,B 0,C 180,E1 3050.789,E2 3050.789} C_VEL
LIN {X 0,Y 103.738,Z 432.276,A -85,B 0,C 180,E1 3053.049,E2 3053.049} C_VEL
LIN {X 0,Y 114.409,Z 421.381,A -85,B 0,C 180,E1 3055.002,E2 3055.002} C_VEL
LIN {X 0,Y 123.552,Z 409.34,A -85,B 0,C 180,E1 3056.506,E2 3056.506} C_VEL
LIN {X 0,Y 130.586,Z 397.389,A -85,B 0,C 180,E1 3057.599,E2 3057.599} C_VEL
LIN {X 0,Y 133.749,Z 390.769,A -85,B 0,C 180,E1 3058.095,E2 3058.095} C_VEL
LIN {X 0,Y 126.512,Z 404.655,A -85,B 0,C 180,E1 3058.56,E2 3058.56} C_VEL
LIN {X 0,Y 117.232,Z 418.096,A -85,B 0,C 180,E1 3059.285,E2 3059.285} C_VEL
LIN {X 0,Y 111.632,Z 424.7,A -85,B 0,C 180,E1 3059.293,E2 3059.293} C_VEL
LIN {X 0,Y 103.793,Z 432.435,A -85,B 0,C 180,E1 3058.243,E2 3058.243} C_VEL
LIN {X 0,Y 92.41,Z 441.49,A -85,B 0,C 180,E1 3055.817,E2 3055.817} C_VEL
LIN {X 0,Y 88.371,Z 444.21,A -85,B 0,C 180,E1 3054.991,E2 3054.991} C_VEL
LIN {X 0,Y 75.678,Z 451.424,A -85,B 0,C 180,E1 3052.217,E2 3052.217} C_VEL
LIN {X 0,Y 62.301,Z 457.008,A -85,B 0,C 180,E1 3048.191,E2 3048.191} C_VEL
LIN {X 0,Y 49.337,Z 460.726,A -85,B 0,C 180,E1 3042.237,E2 3042.237} C_VEL
LIN {X 0,Y 36.352,Z 462.847,A -85,B 0,C 180,E1 3031.635,E2 3031.635} C_VEL
LIN {X 0,Y 25.045,Z 463.076,A -85,B 0,C 180,E1 3009.675,E2 3009.675} C_VEL
LIN {X 0,Y 20.738,Z 461.426,A -85,B 0,C 180,E1 2972.742,E2 2972.742} C_VEL
LIN {X 0,Y 22.553,Z 459.713,A -85,B 0,C 180,E1 2950.558,E2 2950.558} C_VEL
LIN {X 0,Y 22.978,Z 457.937,A -85,B 0,C 180,E1 2902.334,E2 2902.334} C_VEL
LIN {X 0,Y 35.087,Z 462.908,A -85,B 0,C 180,E1 2876.019,E2 2876.019} C_VEL
LIN {X 0,Y 42.478,Z 464.672,A -85,B 0,C 180,E1 2869.149,E2 2869.149} C_VEL
LIN {X 0,Y 25.924,Z 463.333,A -85,B 0,C 180,E1 2848.082,E2 2848.082} C_VEL
LIN {X 0,Y 22.796,Z 462.806,A -85,B 0,C 180,E1 2838.242,E2 2838.242} C_VEL
LIN {X 0,Y 18.653,Z 466.709,A -85,B 0,C 180,E1 2796.178,E2 2796.178} C_VEL
LIN {X 0,Y 18.773,Z 467.046,A -85,B 0,C 180,E1 2790.023,E2 2790.023} C_VEL
LIN {X 0,Y 20.903,Z 467.768,A -85,B 0,C 180,E1 2744.184,E2 2744.184} C_VEL
LIN {X 0,Y 32.622,Z 466.601,A -85,B 0,C 180,E1 2718.215,E2 2718.215} C_VEL
LIN {X 0,Y 47.461,Z 463.382,A -85,B 0,C 180,E1 2707.259,E2 2707.259} C_VEL
LIN {X 0,Y 63.017,Z 458.071,A -85,B 0,C 180,E1 2701.891,E2 2701.891} C_VEL
LIN {X 0,Y 76.989,Z 451.399,A -85,B 0,C 180,E1 2699.117,E2 2699.117} C_VEL
LIN {X 0,Y 90.07,Z 443.269,A -85,B 0,C 180,E1 2697.417,E2 2697.417} C_VEL
LIN {X 0,Y 97.864,Z 437.395,A -85,B 0,C 180,E1 2696.659,E2 2696.659} C_VEL
LIN {X 0,Y 88.371,Z 444.21,A -85,B 0,C 180,E1 2694.991,E2 2694.991} C_VEL
LIN {X 0,Y 80.099,Z 449.19,A -85,B 0,C 180,E1 2694.001,E2 2694.001} C_VEL
LIN {X 0,Y 66.903,Z 455.663,A -85,B 0,C 180,E1 2693.776,E2 2693.776} C_VEL
LIN {X 0,Y 55.085,Z 459.892,A -85,B 0,C 180,E1 2693.254,E2 2693.254} C_VEL
LIN {X 0,Y 47.806,Z 461.685,A -85,B 0,C 180,E1 2691.572,E2 2691.572} C_VEL
LIN {X 0,Y 33.305,Z 463.909,A -85,B 0,C 180,E1 2683.828,E2 2683.828} C_VEL
LIN {X 0,Y 20.34,Z 464.217,A -85,B 0,C 180,E1 2666.646,E2 2666.646} C_VEL
LIN {X 0,Y 12.942,Z 462.916,A -85,B 0,C 180,E1 2623.366,E2 2623.366} C_VEL
LIN {X 0,Y 13.972,Z 461.461,A -85,B 0,C 180,E1 2588.501,E2 2588.501} C_VEL
LIN {X 0,Y 19.731,Z 459.802,A -85,B 0,C 180,E1 2519.177,E2 2519.177} C_VEL
LIN {X 0,Y 25.448,Z 461.881,A -85,B 0,C 180,E1 2509.281,E2 2509.281} C_VEL
LIN {X 0,Y 19.246,Z 461.174,A -85,B 0,C 180,E1 2499.307,E2 2499.307} C_VEL
LIN {X 0,Y 10.596,Z 465.316,A -85,B 0,C 180,E1 2446.488,E2 2446.488} C_VEL
LIN {X 0,Y 10.596,Z 465.851,A -85,B 0,C 180,E1 2430.041,E2 2430.041} C_VEL
LIN {X 0,Y 16.278,Z 466.624,A -85,B 0,C 180,E1 2362.949,E2 2362.949} C_VEL
LIN {X 0,Y 31.049,Z 465.506,A -85,B 0,C 180,E1 2343.619,E2 2343.619} C_VEL
LIN {X 0,Y 47.037,Z 462.36,A -85,B 0,C 180,E1 2337.307,E2 2337.307} C_VEL
LIN {X 0,Y 58.982,Z 458.709,A -85,B 0,C 180,E1 2335.009,E2 2335.009} C_VEL
LIN {X 0,Y 47.806,Z 461.685,A -85,B 0,C 180,E1 2331.572,E2 2331.572} C_VEL
LIN {X 0,Y 39.238,Z 463.328,A -85,B 0,C 180,E1 2329.245,E2 2329.245} C_VEL
LIN {X 0,Y 25.325,Z 464.936,A -85,B 0,C 180,E1 2327.478,E2 2327.478} C_VEL
LIN {X 0,Y 13.963,Z 465.096,A -85,B 0,C 180,E1 2322.76,E2 2322.76} C_VEL
LIN {X 0,Y 8.205,Z 464.585,A -85,B 0,C 180,E1 2308.699,E2 2308.699} C_VEL
LIN {X 0,Y 5.548,Z 463.185,A -85,B 0,C 180,E1 2224.359,E2 2224.359} C_VEL
LIN {X 0,Y 8.539,Z 462.794,A -85,B 0,C 180,E1 2155.055,E2 2155.055} C_VEL
LIN {X 0,Y 2.407,Z 464.655,A -85,B 0,C 180,E1 2070.181,E2 2070.181} C_VEL
LIN {X 0,Y 15.563,Z 465.47,A -85,B 0,C 180,E1 1972.61,E2 1972.61} C_VEL
LIN {X 0,Y 18.954,Z 465.382,A -85,B 0,C 180,E1 1970.888,E2 1970.888} C_VEL
LIN {X 0,Y 8.205,Z 464.585,A -85,B 0,C 180,E1 1948.699,E2 1948.699} C_VEL
LIN {X 0,Y 6.554,Z 466.571,A -85,B 0,C 180,E1 1936.891,E2 1936.891} C_VEL
LIN {X 0,Y 6.554,Z 550,A -85,B 0,C 180,E1 1936.891,E2 1936.891} C_VEL
LIN {X 0,Y 6.554,Z 550,A -85,B 0,C 180,E1 1936.891,E2 1936.891}

QRS_NEXT_CUT()

QRS_NEXT()
QRS_HOME()

END
